LIN {X 0,Y 509.993,Z 290.092,A -85,B 0,C 180,E1 -5500.32,E2 -5500.32} C_VEL
LIN {X 0,Y 510.308,Z 281.912,A -85,B 0,C 180,E1 -5501.117,E2 -5501.117} C_VEL
LIN {X 0,Y 510.541,Z 273.397,A -85,B 0,C 180,E1 -5501.816,E2 -5501.816} C_VEL
LIN {X 0,Y 510.81,Z 263.864,A -85,B 0,C 180,E1 -5502.464,E2 -5502.464} C_VEL
LIN {X 0,Y 511.035,Z 254.914,A -85,B 0,C 180,E1 -5502.964,E2 -5502.964} C_VEL
LIN {X 0,Y 511.335,Z 244.83,A -85,B 0,C 180,E1 -5503.411,E2 -5503.411} C_VEL
LIN {X 0,Y 511.524,Z 235.312,A -85,B 0,C 180,E1 -5503.735,E2 -5503.735} C_VEL
LIN {X 0,Y 511.735,Z 224.998,A -85,B 0,C 180,E1 -5503.983,E2 -5503.983} C_VEL
LIN {X 0,Y 512.09,Z 160.549,A -85,B 0,C 180,E1 -5504.912,E2 -5504.912} C_VEL
LIN {X 0,Y 512.087,Z 131.63,A -85,B 0,C 180,E1 -5505.323,E2 -5505.323} C_VEL
LIN {X 0,Y 510.005,Z 119.074,A -85,B 0,C 180,E1 -5505.584,E2 -5505.584} C_VEL
LIN {X 0,Y 509.995,Z 117.671,A -85,B 0,C 180,E1 -5505.801,E2 -5505.801} C_VEL
LIN {X 0,Y 510.345,Z 103.483,A -85,B 0,C 180,E1 -5508.674,E2 -5508.674} C_VEL
LIN {X 0,Y 510.685,Z 89.891,A -85,B 0,C 180,E1 -5511.388,E2 -5511.388} C_VEL
LIN {X 0,Y 511.184,Z 75.466,A -85,B 0,C 180,E1 -5514.359,E2 -5514.359} C_VEL
LIN {X 0,Y 510.796,Z 71.345,A -85,B 0,C 180,E1 -5515.247,E2 -5515.247} C_VEL
LIN {X 0,Y 509.918,Z 66.493,A -85,B 0,C 180,E1 -5516.379,E2 -5516.379} C_VEL
LIN {X 0,Y 509.88,Z 66.471,A -85,B 0,C 180,E1 -5518.844,E2 -5518.844} C_VEL
LIN {X 0,Y 509.823,Z 66.48,A -85,B 0,C 180,E1 -5521.59,E2 -5521.59} C_VEL
LIN {X 0,Y 509.855,Z 66.471,A -85,B 0,C 180,E1 -5524.413,E2 -5524.413} C_VEL
LIN {X 0,Y 509.82,Z 66.479,A -85,B 0,C 180,E1 -5527.34,E2 -5527.34} C_VEL
LIN {X 0,Y 509.84,Z 66.466,A -85,B 0,C 180,E1 -5530.382,E2 -5530.382} C_VEL
LIN {X 0,Y 509.824,Z 66.478,A -85,B 0,C 180,E1 -5533.062,E2 -5533.062} C_VEL
LIN {X 0,Y 509.824,Z 66.478,A -85,B 0,C 180,E1 -5535.793,E2 -5535.793} C_VEL
LIN {X 0,Y 509.857,Z 66.471,A -85,B 0,C 180,E1 -5538.574,E2 -5538.574} C_VEL
LIN {X 0,Y 509.853,Z 66.473,A -85,B 0,C 180,E1 -5541.786,E2 -5541.786} C_VEL
LIN {X 0,Y 509.835,Z 66.474,A -85,B 0,C 180,E1 -5544.622,E2 -5544.622} C_VEL
LIN {X 0,Y 509.862,Z 66.472,A -85,B 0,C 180,E1 -5547.48,E2 -5547.48} C_VEL
LIN {X 0,Y 509.86,Z 66.471,A -85,B 0,C 180,E1 -5550.273,E2 -5550.273} C_VEL
LIN {X 0,Y 509.885,Z 66.466,A -85,B 0,C 180,E1 -5552.944,E2 -5552.944} C_VEL
LIN {X 0,Y 509.871,Z 66.468,A -85,B 0,C 180,E1 -5555.574,E2 -5555.574} C_VEL
LIN {X 0,Y 509.852,Z 66.47,A -85,B 0,C 180,E1 -5558.998,E2 -5558.998} C_VEL
LIN {X 0,Y 509.883,Z 66.459,A -85,B 0,C 180,E1 -5562.001,E2 -5562.001} C_VEL
LIN {X 0,Y 509.911,Z 66.467,A -85,B 0,C 180,E1 -5564.818,E2 -5564.818} C_VEL
LIN {X 0,Y 509.902,Z 66.468,A -85,B 0,C 180,E1 -5568.123,E2 -5568.123} C_VEL
LIN {X 0,Y 509.915,Z 66.455,A -85,B 0,C 180,E1 -5571.279,E2 -5571.279} C_VEL
LIN {X 0,Y 509.979,Z 66.455,A -85,B 0,C 180,E1 -5573.67,E2 -5573.67} C_VEL
LIN {X 0,Y 510.055,Z 66.447,A -85,B 0,C 180,E1 -5577.63,E2 -5577.63} C_VEL
LIN {X 0,Y 510.063,Z 66.436,A -85,B 0,C 180,E1 -5580.789,E2 -5580.789} C_VEL
LIN {X 0,Y 509.953,Z 66.457,A -85,B 0,C 180,E1 -5583.16,E2 -5583.16} C_VEL
LIN {X 0,Y 509.978,Z 66.455,A -85,B 0,C 180,E1 -5586.329,E2 -5586.329} C_VEL
LIN {X 0,Y 509.914,Z 66.456,A -85,B 0,C 180,E1 -5588.72,E2 -5588.72} C_VEL
LIN {X 0,Y 509.951,Z 66.46,A -85,B 0,C 180,E1 -5591.93,E2 -5591.93} C_VEL
LIN {X 0,Y 509.893,Z 66.472,A -85,B 0,C 180,E1 -5595.241,E2 -5595.241} C_VEL
LIN {X 0,Y 509.887,Z 66.46,A -85,B 0,C 180,E1 -5598,E2 -5598} C_VEL
LIN {X 0,Y 509.849,Z 66.471,A -85,B 0,C 180,E1 -5601.001,E2 -5601.001} C_VEL
LIN {X 0,Y 509.868,Z 66.47,A -85,B 0,C 180,E1 -5604.426,E2 -5604.426} C_VEL
LIN {X 0,Y 509.883,Z 66.466,A -85,B 0,C 180,E1 -5607.055,E2 -5607.055} C_VEL
LIN {X 0,Y 509.855,Z 66.471,A -85,B 0,C 180,E1 -5609.751,E2 -5609.751} C_VEL
LIN {X 0,Y 509.874,Z 66.475,A -85,B 0,C 180,E1 -5612.774,E2 -5612.774} C_VEL
LIN {X 0,Y 509.84,Z 66.471,A -85,B 0,C 180,E1 -5615.581,E2 -5615.581} C_VEL
LIN {X 0,Y 509.848,Z 66.476,A -85,B 0,C 180,E1 -5618.338,E2 -5618.338} C_VEL
LIN {X 0,Y 509.862,Z 66.468,A -85,B 0,C 180,E1 -5621.424,E2 -5621.424} C_VEL
LIN {X 0,Y 509.854,Z 66.474,A -85,B 0,C 180,E1 -5624.668,E2 -5624.668} C_VEL
LIN {X 0,Y 509.855,Z 66.46,A -85,B 0,C 180,E1 -5628.103,E2 -5628.103} C_VEL
LIN {X 0,Y 509.844,Z 66.476,A -85,B 0,C 180,E1 -5630.648,E2 -5630.648} C_VEL
LIN {X 0,Y 509.829,Z 66.474,A -85,B 0,C 180,E1 -5633.732,E2 -5633.732} C_VEL
LIN {X 0,Y 509.163,Z 66.553,A -85,B 0,C 180,E1 -5634.391,E2 -5634.391} C_VEL
LIN {X 0,Y 506.346,Z 66.901,A -85,B 0,C 180,E1 -5635.463,E2 -5635.463} C_VEL
LIN {X 0,Y 503.953,Z 67.206,A -85,B 0,C 180,E1 -5636.327,E2 -5636.327} C_VEL
LIN {X 0,Y 502.903,Z 67.336,A -85,B 0,C 180,E1 -5636.993,E2 -5636.993} C_VEL
LIN {X 0,Y 502.806,Z 67.348,A -85,B 0,C 180,E1 -5637.219,E2 -5637.219} C_VEL
LIN {X 0,Y 502.811,Z 67.347,A -85,B 0,C 180,E1 -5640.065,E2 -5640.065} C_VEL
LIN {X 0,Y 502.831,Z 67.349,A -85,B 0,C 180,E1 -5642.533,E2 -5642.533} C_VEL
LIN {X 0,Y 502.826,Z 67.35,A -85,B 0,C 180,E1 -5645.298,E2 -5645.298} C_VEL
LIN {X 0,Y 502.782,Z 67.36,A -85,B 0,C 180,E1 -5647.827,E2 -5647.827} C_VEL
LIN {X 0,Y 502.822,Z 67.35,A -85,B 0,C 180,E1 -5650.4,E2 -5650.4} C_VEL
LIN {X 0,Y 502.831,Z 67.349,A -85,B 0,C 180,E1 -5652.932,E2 -5652.932} C_VEL
LIN {X 0,Y 502.849,Z 67.352,A -85,B 0,C 180,E1 -5655.429,E2 -5655.429} C_VEL
LIN {X 0,Y 502.874,Z 67.344,A -85,B 0,C 180,E1 -5658.717,E2 -5658.717} C_VEL
LIN {X 0,Y 502.899,Z 67.341,A -85,B 0,C 180,E1 -5661.967,E2 -5661.967} C_VEL
LIN {X 0,Y 502.939,Z 67.336,A -85,B 0,C 180,E1 -5664.387,E2 -5664.387} C_VEL
LIN {X 0,Y 503.023,Z 67.327,A -85,B 0,C 180,E1 -5667.598,E2 -5667.598} C_VEL
LIN {X 0,Y 503.025,Z 67.325,A -85,B 0,C 180,E1 -5670,E2 -5670} C_VEL
LIN {X 0,Y 503.023,Z 67.326,A -85,B 0,C 180,E1 -5672.402,E2 -5672.402} C_VEL
LIN {X 0,Y 502.939,Z 67.336,A -85,B 0,C 180,E1 -5675.613,E2 -5675.613} C_VEL
LIN {X 0,Y 502.899,Z 67.341,A -85,B 0,C 180,E1 -5678.033,E2 -5678.033} C_VEL
LIN {X 0,Y 502.874,Z 67.344,A -85,B 0,C 180,E1 -5681.283,E2 -5681.283} C_VEL
LIN {X 0,Y 502.849,Z 67.352,A -85,B 0,C 180,E1 -5684.571,E2 -5684.571} C_VEL
LIN {X 0,Y 502.859,Z 67.347,A -85,B 0,C 180,E1 -5687.907,E2 -5687.907} C_VEL
LIN {X 0,Y 502.825,Z 67.354,A -85,B 0,C 180,E1 -5690.536,E2 -5690.536} C_VEL
LIN {X 0,Y 502.794,Z 67.353,A -85,B 0,C 180,E1 -5693.04,E2 -5693.04} C_VEL
LIN {X 0,Y 502.837,Z 67.349,A -85,B 0,C 180,E1 -5695.676,E2 -5695.676} C_VEL
LIN {X 0,Y 502.837,Z 67.344,A -85,B 0,C 180,E1 -5698.373,E2 -5698.373} C_VEL
LIN {X 0,Y 502.793,Z 67.353,A -85,B 0,C 180,E1 -5701.5,E2 -5701.5} C_VEL
LIN {X 0,Y 502.803,Z 67.337,A -85,B 0,C 180,E1 -5704.445,E2 -5704.445} C_VEL
LIN {X 0,Y 502.778,Z 67.353,A -85,B 0,C 180,E1 -5707.179,E2 -5707.179} C_VEL
LIN {X 0,Y 502.785,Z 67.348,A -85,B 0,C 180,E1 -5710.015,E2 -5710.015} C_VEL
LIN {X 0,Y 502.799,Z 67.336,A -85,B 0,C 180,E1 -5712.199,E2 -5712.199} C_VEL
LIN {X 0,Y 502.798,Z 67.354,A -85,B 0,C 180,E1 -5715.468,E2 -5715.468} C_VEL
LIN {X 0,Y 502.823,Z 67.348,A -85,B 0,C 180,E1 -5719.004,E2 -5719.004} C_VEL
LIN {X 0,Y 502.791,Z 67.352,A -85,B 0,C 180,E1 -5722.047,E2 -5722.047} C_VEL
LIN {X 0,Y 502.807,Z 67.35,A -85,B 0,C 180,E1 -5725.035,E2 -5725.035} C_VEL
LIN {X 0,Y 502.782,Z 67.352,A -85,B 0,C 180,E1 -5727.916,E2 -5727.916} C_VEL
LIN {X 0,Y 502.822,Z 67.351,A -85,B 0,C 180,E1 -5730.713,E2 -5730.713} C_VEL
LIN {X 0,Y 502.86,Z 67.339,A -85,B 0,C 180,E1 -5733.44,E2 -5733.44} C_VEL
LIN {X 0,Y 502.79,Z 67.351,A -85,B 0,C 180,E1 -5736.087,E2 -5736.087} C_VEL
LIN {X 0,Y 502.782,Z 67.356,A -85,B 0,C 180,E1 -5738.689,E2 -5738.689} C_VEL
LIN {X 0,Y 502.829,Z 67.339,A -85,B 0,C 180,E1 -5741.249,E2 -5741.249} C_VEL
LIN {X 0,Y 502.821,Z 67.345,A -85,B 0,C 180,E1 -5743.768,E2 -5743.768} C_VEL
LIN {X 0,Y 502.83,Z 67.351,A -85,B 0,C 180,E1 -5746.255,E2 -5746.255} C_VEL
LIN {X 0,Y 502.892,Z 67.333,A -85,B 0,C 180,E1 -5748.718,E2 -5748.718} C_VEL
LIN {X 0,Y 502.901,Z 67.333,A -85,B 0,C 180,E1 -5751.967,E2 -5751.967} C_VEL
LIN {X 0,Y 502.937,Z 67.339,A -85,B 0,C 180,E1 -5754.387,E2 -5754.387} C_VEL
LIN {X 0,Y 503.024,Z 67.321,A -85,B 0,C 180,E1 -5757.598,E2 -5757.598} C_VEL
LIN {X 0,Y 503.027,Z 67.315,A -85,B 0,C 180,E1 -5760,E2 -5760} C_VEL
LIN {X 0,Y 503.025,Z 67.322,A -85,B 0,C 180,E1 -5762.403,E2 -5762.403} C_VEL
LIN {X 0,Y 502.938,Z 67.338,A -85,B 0,C 180,E1 -5765.614,E2 -5765.614} C_VEL
LIN {X 0,Y 502.902,Z 67.333,A -85,B 0,C 180,E1 -5768.034,E2 -5768.034} C_VEL
LIN {X 0,Y 502.878,Z 67.334,A -85,B 0,C 180,E1 -5771.284,E2 -5771.284} C_VEL
LIN {X 0,Y 502.846,Z 67.343,A -85,B 0,C 180,E1 -5774.571,E2 -5774.571} C_VEL
LIN {X 0,Y 502.856,Z 67.334,A -85,B 0,C 180,E1 -5777.908,E2 -5777.908} C_VEL
LIN {X 0,Y 502.83,Z 67.341,A -85,B 0,C 180,E1 -5780.537,E2 -5780.537} C_VEL
LIN {X 0,Y 502.796,Z 67.354,A -85,B 0,C 180,E1 -5783.041,E2 -5783.041} C_VEL
LIN {X 0,Y 502.841,Z 67.34,A -85,B 0,C 180,E1 -5785.676,E2 -5785.676} C_VEL
LIN {X 0,Y 502.841,Z 67.34,A -85,B 0,C 180,E1 -5788.373,E2 -5788.373} C_VEL
LIN {X 0,Y 502.794,Z 67.352,A -85,B 0,C 180,E1 -5791.499,E2 -5791.499} C_VEL
LIN {X 0,Y 502.807,Z 67.342,A -85,B 0,C 180,E1 -5793.994,E2 -5793.994} C_VEL
LIN {X 0,Y 502.779,Z 67.356,A -85,B 0,C 180,E1 -5797.178,E2 -5797.178} C_VEL
LIN {X 0,Y 502.789,Z 67.348,A -85,B 0,C 180,E1 -5800.016,E2 -5800.016} C_VEL
LIN {X 0,Y 502.804,Z 67.352,A -85,B 0,C 180,E1 -5802.2,E2 -5802.2} C_VEL
LIN {X 0,Y 502.787,Z 67.35,A -85,B 0,C 180,E1 -5805.47,E2 -5805.47} C_VEL
LIN {X 0,Y 502.821,Z 67.341,A -85,B 0,C 180,E1 -5808.934,E2 -5808.934} C_VEL
LIN {X 0,Y 502.795,Z 67.354,A -85,B 0,C 180,E1 -5812.046,E2 -5812.046} C_VEL
LIN {X 0,Y 502.81,Z 67.347,A -85,B 0,C 180,E1 -5815.035,E2 -5815.035} C_VEL
LIN {X 0,Y 502.786,Z 67.354,A -85,B 0,C 180,E1 -5817.916,E2 -5817.916} C_VEL
LIN {X 0,Y 502.827,Z 67.35,A -85,B 0,C 180,E1 -5820.712,E2 -5820.712} C_VEL
LIN {X 0,Y 502.899,Z 67.568,A -85,B 0,C 180,E1 -5823.524,E2 -5823.524} C_VEL
LIN {X 0,Y 504.176,Z 75.331,A -85,B 0,C 180,E1 -5825.28,E2 -5825.28} C_VEL
LIN {X 0,Y 503.8,Z 87.666,A -85,B 0,C 180,E1 -5827.874,E2 -5827.874} C_VEL
LIN {X 0,Y 503.438,Z 101.167,A -85,B 0,C 180,E1 -5830.637,E2 -5830.637} C_VEL
LIN {X 0,Y 503.066,Z 114.588,A -85,B 0,C 180,E1 -5833.358,E2 -5833.358} C_VEL
LIN {X 0,Y 502.97,Z 118.697,A -85,B 0,C 180,E1 -5834.179,E2 -5834.179} C_VEL
LIN {X 0,Y 504.693,Z 129.277,A -85,B 0,C 180,E1 -5834.416,E2 -5834.416} C_VEL
LIN {X 0,Y 505.338,Z 134.211,A -85,B 0,C 180,E1 -5834.507,E2 -5834.507} C_VEL
LIN {X 0,Y 504.875,Z 223.476,A -85,B 0,C 180,E1 -5835.798,E2 -5835.798} C_VEL
LIN {X 0,Y 504.64,Z 234.247,A -85,B 0,C 180,E1 -5836.048,E2 -5836.048} C_VEL
LIN {X 0,Y 504.462,Z 243.352,A -85,B 0,C 180,E1 -5836.351,E2 -5836.351} C_VEL
LIN {X 0,Y 504.145,Z 253.716,A -85,B 0,C 180,E1 -5836.805,E2 -5836.805} C_VEL
LIN {X 0,Y 503.863,Z 263.769,A -85,B 0,C 180,E1 -5837.367,E2 -5837.367} C_VEL
LIN {X 0,Y 503.589,Z 271.853,A -85,B 0,C 180,E1 -5837.917,E2 -5837.917} C_VEL
LIN {X 0,Y 503.31,Z 280.584,A -85,B 0,C 180,E1 -5838.625,E2 -5838.625} C_VEL
LIN {X 0,Y 503.05,Z 287.981,A -85,B 0,C 180,E1 -5839.332,E2 -5839.332} C_VEL
LIN {X 0,Y 502.829,Z 295.203,A -85,B 0,C 180,E1 -5840.141,E2 -5840.141} C_VEL
LIN {X 0,Y 502.608,Z 301.404,A -85,B 0,C 180,E1 -5840.949,E2 -5840.949} C_VEL
LIN {X 0,Y 502.425,Z 307.942,A -85,B 0,C 180,E1 -5841.959,E2 -5841.959} C_VEL
LIN {X 0,Y 502.273,Z 313.495,A -85,B 0,C 180,E1 -5842.988,E2 -5842.988} C_VEL
LIN {X 0,Y 502.189,Z 317.931,A -85,B 0,C 180,E1 -5843.975,E2 -5843.975} C_VEL
LIN {X 0,Y 502.11,Z 322.251,A -85,B 0,C 180,E1 -5845.183,E2 -5845.183} C_VEL
LIN {X 0,Y 502.138,Z 324.616,A -85,B 0,C 180,E1 -5845.987,E2 -5845.987} C_VEL
LIN {X 0,Y 502.12,Z 326.411,A -85,B 0,C 180,E1 -5846.791,E2 -5846.791} C_VEL
LIN {X 0,Y 502.037,Z 328.849,A -85,B 0,C 180,E1 -5848.396,E2 -5848.396} C_VEL
LIN {X 0,Y 501.994,Z 329.435,A -85,B 0,C 180,E1 -5849.198,E2 -5849.198} C_VEL
LIN {X 0,Y 501.994,Z 329.435,A -85,B 0,C 180,E1 -5850.802,E2 -5850.802} C_VEL
LIN {X 0,Y 502.037,Z 328.849,A -85,B 0,C 180,E1 -5851.604,E2 -5851.604} C_VEL
LIN {X 0,Y 502.12,Z 326.411,A -85,B 0,C 180,E1 -5853.209,E2 -5853.209} C_VEL
LIN {X 0,Y 502.103,Z 323.466,A -85,B 0,C 180,E1 -5854.415,E2 -5854.415} C_VEL
LIN {X 0,Y 502.194,Z 319.484,A -85,B 0,C 180,E1 -5855.622,E2 -5855.622} C_VEL
LIN {X 0,Y 502.217,Z 314.548,A -85,B 0,C 180,E1 -5856.791,E2 -5856.791} C_VEL
LIN {X 0,Y 502.381,Z 309.097,A -85,B 0,C 180,E1 -5857.839,E2 -5857.839} C_VEL
LIN {X 0,Y 502.572,Z 302.781,A -85,B 0,C 180,E1 -5858.849,E2 -5858.849} C_VEL
LIN {X 0,Y 502.775,Z 296.83,A -85,B 0,C 180,E1 -5859.656,E2 -5859.656} C_VEL
LIN {X 0,Y 502.971,Z 289.9,A -85,B 0,C 180,E1 -5860.466,E2 -5860.466} C_VEL
LIN {X 0,Y 503.268,Z 281.719,A -85,B 0,C 180,E1 -5861.274,E2 -5861.274} C_VEL
LIN {X 0,Y 503.567,Z 273.206,A -85,B 0,C 180,E1 -5861.982,E2 -5861.982} C_VEL
LIN {X 0,Y 503.843,Z 264.07,A -85,B 0,C 180,E1 -5862.615,E2 -5862.615} C_VEL
LIN {X 0,Y 504.09,Z 254.723,A -85,B 0,C 180,E1 -5863.146,E2 -5863.146} C_VEL
LIN {X 0,Y 504.419,Z 244.639,A -85,B 0,C 180,E1 -5863.598,E2 -5863.598} C_VEL
LIN {X 0,Y 504.646,Z 235.122,A -85,B 0,C 180,E1 -5863.926,E2 -5863.926} C_VEL
LIN {X 0,Y 504.848,Z 224.808,A -85,B 0,C 180,E1 -5864.177,E2 -5864.177} C_VEL
LIN {X 0,Y 505.172,Z 165.727,A -85,B 0,C 180,E1 -5865.043,E2 -5865.043} C_VEL
LIN {X 0,Y 505.145,Z 131.725,A -85,B 0,C 180,E1 -5865.534,E2 -5865.534} C_VEL
LIN {X 0,Y 502.987,Z 118.974,A -85,B 0,C 180,E1 -5865.802,E2 -5865.802} C_VEL
LIN {X 0,Y 502.957,Z 117.857,A -85,B 0,C 180,E1 -5865.947,E2 -5865.947} C_VEL
LIN {X 0,Y 503.347,Z 104.398,A -85,B 0,C 180,E1 -5868.732,E2 -5868.732} C_VEL
LIN {X 0,Y 503.695,Z 90.805,A -85,B 0,C 180,E1 -5871.485,E2 -5871.485} C_VEL
LIN {X 0,Y 504.204,Z 77.414,A -85,B 0,C 180,E1 -5874.28,E2 -5874.28} C_VEL
LIN {X 0,Y 503.885,Z 72.915,A -85,B 0,C 180,E1 -5875.259,E2 -5875.259} C_VEL
LIN {X 0,Y 502.885,Z 67.367,A -85,B 0,C 180,E1 -5876.565,E2 -5876.565} C_VEL
LIN {X 0,Y 502.827,Z 67.35,A -85,B 0,C 180,E1 -5879.288,E2 -5879.288} C_VEL
LIN {X 0,Y 502.786,Z 67.355,A -85,B 0,C 180,E1 -5882.084,E2 -5882.084} C_VEL
LIN {X 0,Y 502.81,Z 67.348,A -85,B 0,C 180,E1 -5884.965,E2 -5884.965} C_VEL
LIN {X 0,Y 502.795,Z 67.354,A -85,B 0,C 180,E1 -5887.954,E2 -5887.954} C_VEL
LIN {X 0,Y 502.821,Z 67.342,A -85,B 0,C 180,E1 -5891.066,E2 -5891.066} C_VEL
LIN {X 0,Y 502.787,Z 67.351,A -85,B 0,C 180,E1 -5894.53,E2 -5894.53} C_VEL
LIN {X 0,Y 502.796,Z 67.352,A -85,B 0,C 180,E1 -5897.86,E2 -5897.86} C_VEL
LIN {X 0,Y 502.803,Z 67.351,A -85,B 0,C 180,E1 -5901.024,E2 -5901.024} C_VEL
LIN {X 0,Y 502.778,Z 67.351,A -85,B 0,C 180,E1 -5904.168,E2 -5904.168} C_VEL
LIN {X 0,Y 502.834,Z 67.347,A -85,B 0,C 180,E1 -5906.993,E2 -5906.993} C_VEL
LIN {X 0,Y 502.816,Z 67.348,A -85,B 0,C 180,E1 -5910.065,E2 -5910.065} C_VEL
LIN {X 0,Y 502.833,Z 67.344,A -85,B 0,C 180,E1 -5912.533,E2 -5912.533} C_VEL
LIN {X 0,Y 502.83,Z 67.347,A -85,B 0,C 180,E1 -5915.298,E2 -5915.298} C_VEL
LIN {X 0,Y 502.782,Z 67.351,A -85,B 0,C 180,E1 -5917.826,E2 -5917.826} C_VEL
LIN {X 0,Y 502.826,Z 67.345,A -85,B 0,C 180,E1 -5920.4,E2 -5920.4} C_VEL
LIN {X 0,Y 502.831,Z 67.345,A -85,B 0,C 180,E1 -5922.931,E2 -5922.931} C_VEL
LIN {X 0,Y 502.846,Z 67.343,A -85,B 0,C 180,E1 -5925.429,E2 -5925.429} C_VEL
LIN {X 0,Y 502.878,Z 67.334,A -85,B 0,C 180,E1 -5928.716,E2 -5928.716} C_VEL
LIN {X 0,Y 502.902,Z 67.333,A -85,B 0,C 180,E1 -5931.966,E2 -5931.966} C_VEL
LIN {X 0,Y 502.938,Z 67.338,A -85,B 0,C 180,E1 -5934.386,E2 -5934.386} C_VEL
LIN {X 0,Y 503.025,Z 67.322,A -85,B 0,C 180,E1 -5937.597,E2 -5937.597} C_VEL
LIN {X 0,Y 503.027,Z 67.315,A -85,B 0,C 180,E1 -5940,E2 -5940} C_VEL
LIN {X 0,Y 503.024,Z 67.321,A -85,B 0,C 180,E1 -5942.402,E2 -5942.402} C_VEL
LIN {X 0,Y 502.937,Z 67.339,A -85,B 0,C 180,E1 -5945.613,E2 -5945.613} C_VEL
LIN {X 0,Y 502.901,Z 67.333,A -85,B 0,C 180,E1 -5948.033,E2 -5948.033} C_VEL
LIN {X 0,Y 502.892,Z 67.333,A -85,B 0,C 180,E1 -5951.282,E2 -5951.282} C_VEL
LIN {X 0,Y 502.844,Z 67.344,A -85,B 0,C 180,E1 -5954.57,E2 -5954.57} C_VEL
LIN {X 0,Y 502.86,Z 67.335,A -85,B 0,C 180,E1 -5957.907,E2 -5957.907} C_VEL
LIN {X 0,Y 502.827,Z 67.341,A -85,B 0,C 180,E1 -5960.536,E2 -5960.536} C_VEL
LIN {X 0,Y 502.793,Z 67.356,A -85,B 0,C 180,E1 -5963.04,E2 -5963.04} C_VEL
LIN {X 0,Y 502.838,Z 67.342,A -85,B 0,C 180,E1 -5965.675,E2 -5965.675} C_VEL
LIN {X 0,Y 502.838,Z 67.34,A -85,B 0,C 180,E1 -5968.372,E2 -5968.372} C_VEL
LIN {X 0,Y 502.794,Z 67.352,A -85,B 0,C 180,E1 -5971.499,E2 -5971.499} C_VEL
LIN {X 0,Y 502.804,Z 67.348,A -85,B 0,C 180,E1 -5974.444,E2 -5974.444} C_VEL
LIN {X 0,Y 502.778,Z 67.356,A -85,B 0,C 180,E1 -5977.178,E2 -5977.178} C_VEL
LIN {X 0,Y 502.814,Z 67.347,A -85,B 0,C 180,E1 -5980.012,E2 -5980.012} C_VEL
LIN {X 0,Y 502.77,Z 67.355,A -85,B 0,C 180,E1 -5983.231,E2 -5983.231} C_VEL
LIN {X 0,Y 502.786,Z 67.348,A -85,B 0,C 180,E1 -5985.661,E2 -5985.661} C_VEL
LIN {X 0,Y 502.816,Z 67.341,A -85,B 0,C 180,E1 -5989.005,E2 -5989.005} C_VEL
LIN {X 0,Y 502.791,Z 67.357,A -85,B 0,C 180,E1 -5992.046,E2 -5992.046} C_VEL
LIN {X 0,Y 502.807,Z 67.338,A -85,B 0,C 180,E1 -5995.035,E2 -5995.035} C_VEL
LIN {X 0,Y 502.806,Z 67.348,A -85,B 0,C 180,E1 -5997.219,E2 -5997.219} C_VEL
LIN {X 0,Y 502.104,Z 67.443,A -85,B 0,C 180,E1 -5997.888,E2 -5997.888} C_VEL
LIN {X 0,Y 499.239,Z 67.794,A -85,B 0,C 180,E1 -5998.973,E2 -5998.973} C_VEL
LIN {X 0,Y 496.844,Z 68.093,A -85,B 0,C 180,E1 -5999.848,E2 -5999.848} C_VEL
LIN {X 0,Y 495.828,Z 68.213,A -85,B 0,C 180,E1 -6000.524,E2 -6000.524} C_VEL
LIN {X 0,Y 495.75,Z 68.221,A -85,B 0,C 180,E1 -6000.753,E2 -6000.753} C_VEL
LIN {X 0,Y 495.82,Z 68.222,A -85,B 0,C 180,E1 -6003.251,E2 -6003.251} C_VEL
LIN {X 0,Y 495.75,Z 68.236,A -85,B 0,C 180,E1 -6005.725,E2 -6005.725} C_VEL
LIN {X 0,Y 495.741,Z 68.232,A -85,B 0,C 180,E1 -6008.371,E2 -6008.371} C_VEL
LIN {X 0,Y 495.781,Z 68.227,A -85,B 0,C 180,E1 -6010.972,E2 -6010.972} C_VEL
LIN {X 0,Y 495.776,Z 68.233,A -85,B 0,C 180,E1 -6013.53,E2 -6013.53} C_VEL
LIN {X 0,Y 495.795,Z 68.226,A -85,B 0,C 180,E1 -6016.056,E2 -6016.056} C_VEL
LIN {X 0,Y 495.849,Z 68.219,A -85,B 0,C 180,E1 -6018.555,E2 -6018.555} C_VEL
LIN {X 0,Y 495.87,Z 68.218,A -85,B 0,C 180,E1 -6021.852,E2 -6021.852} C_VEL
LIN {X 0,Y 495.896,Z 68.213,A -85,B 0,C 180,E1 -6024.307,E2 -6024.307} C_VEL
LIN {X 0,Y 495.991,Z 68.203,A -85,B 0,C 180,E1 -6027.564,E2 -6027.564} C_VEL
LIN {X 0,Y 495.996,Z 68.201,A -85,B 0,C 180,E1 -6030,E2 -6030} C_VEL
LIN {X 0,Y 495.991,Z 68.203,A -85,B 0,C 180,E1 -6032.436,E2 -6032.436} C_VEL
LIN {X 0,Y 495.896,Z 68.213,A -85,B 0,C 180,E1 -6035.693,E2 -6035.693} C_VEL
LIN {X 0,Y 495.87,Z 68.218,A -85,B 0,C 180,E1 -6038.148,E2 -6038.148} C_VEL
LIN {X 0,Y 495.849,Z 68.219,A -85,B 0,C 180,E1 -6041.445,E2 -6041.445} C_VEL
LIN {X 0,Y 495.791,Z 68.23,A -85,B 0,C 180,E1 -6044.783,E2 -6044.783} C_VEL
LIN {X 0,Y 495.783,Z 68.226,A -85,B 0,C 180,E1 -6047.319,E2 -6047.319} C_VEL
LIN {X 0,Y 495.775,Z 68.23,A -85,B 0,C 180,E1 -6049.89,E2 -6049.89} C_VEL
LIN {X 0,Y 495.762,Z 68.23,A -85,B 0,C 180,E1 -6052.863,E2 -6052.863} C_VEL
LIN {X 0,Y 495.788,Z 68.231,A -85,B 0,C 180,E1 -6056.068,E2 -6056.068} C_VEL
LIN {X 0,Y 495.769,Z 68.22,A -85,B 0,C 180,E1 -6058.815,E2 -6058.815} C_VEL
LIN {X 0,Y 495.756,Z 68.233,A -85,B 0,C 180,E1 -6061.726,E2 -6061.726} C_VEL
LIN {X 0,Y 495.773,Z 68.211,A -85,B 0,C 180,E1 -6064.695,E2 -6064.695} C_VEL
LIN {X 0,Y 495.729,Z 68.236,A -85,B 0,C 180,E1 -6067.562,E2 -6067.562} C_VEL
LIN {X 0,Y 495.763,Z 68.218,A -85,B 0,C 180,E1 -6070.7,E2 -6070.7} C_VEL
LIN {X 0,Y 495.729,Z 68.229,A -85,B 0,C 180,E1 -6074.001,E2 -6074.001} C_VEL
LIN {X 0,Y 495.723,Z 68.236,A -85,B 0,C 180,E1 -6077.117,E2 -6077.117} C_VEL
LIN {X 0,Y 495.782,Z 68.223,A -85,B 0,C 180,E1 -6079.95,E2 -6079.95} C_VEL
LIN {X 0,Y 495.728,Z 68.232,A -85,B 0,C 180,E1 -6082.553,E2 -6082.553} C_VEL
LIN {X 0,Y 495.783,Z 68.223,A -85,B 0,C 180,E1 -6085.458,E2 -6085.458} C_VEL
LIN {X 0,Y 495.754,Z 68.228,A -85,B 0,C 180,E1 -6088.364,E2 -6088.364} C_VEL
LIN {X 0,Y 495.786,Z 68.219,A -85,B 0,C 180,E1 -6091.507,E2 -6091.507} C_VEL
LIN {X 0,Y 495.789,Z 68.218,A -85,B 0,C 180,E1 -6093.933,E2 -6093.933} C_VEL
LIN {X 0,Y 495.76,Z 68.23,A -85,B 0,C 180,E1 -6097.139,E2 -6097.139} C_VEL
LIN {X 0,Y 495.77,Z 68.221,A -85,B 0,C 180,E1 -6100.11,E2 -6100.11} C_VEL
LIN {X 0,Y 495.786,Z 68.224,A -85,B 0,C 180,E1 -6102.682,E2 -6102.682} C_VEL
LIN {X 0,Y 495.789,Z 68.224,A -85,B 0,C 180,E1 -6105.218,E2 -6105.218} C_VEL
LIN {X 0,Y 495.867,Z 68.21,A -85,B 0,C 180,E1 -6108.556,E2 -6108.556} C_VEL
LIN {X 0,Y 495.872,Z 68.207,A -85,B 0,C 180,E1 -6111.852,E2 -6111.852} C_VEL
LIN {X 0,Y 495.895,Z 68.217,A -85,B 0,C 180,E1 -6114.307,E2 -6114.307} C_VEL
LIN {X 0,Y 495.993,Z 68.197,A -85,B 0,C 180,E1 -6117.564,E2 -6117.564} C_VEL
LIN {X 0,Y 495.983,Z 68.19,A -85,B 0,C 180,E1 -6120.812,E2 -6120.812} C_VEL
LIN {X 0,Y 495.993,Z 68.198,A -85,B 0,C 180,E1 -6122.437,E2 -6122.437} C_VEL
LIN {X 0,Y 495.896,Z 68.216,A -85,B 0,C 180,E1 -6125.694,E2 -6125.694} C_VEL
LIN {X 0,Y 495.873,Z 68.206,A -85,B 0,C 180,E1 -6128.148,E2 -6128.148} C_VEL
LIN {X 0,Y 495.852,Z 68.211,A -85,B 0,C 180,E1 -6131.446,E2 -6131.446} C_VEL
LIN {X 0,Y 495.791,Z 68.222,A -85,B 0,C 180,E1 -6134.783,E2 -6134.783} C_VEL
LIN {X 0,Y 495.783,Z 68.224,A -85,B 0,C 180,E1 -6137.319,E2 -6137.319} C_VEL
LIN {X 0,Y 495.772,Z 68.222,A -85,B 0,C 180,E1 -6139.891,E2 -6139.891} C_VEL
LIN {X 0,Y 495.763,Z 68.228,A -85,B 0,C 180,E1 -6142.862,E2 -6142.862} C_VEL
LIN {X 0,Y 495.792,Z 68.216,A -85,B 0,C 180,E1 -6146.068,E2 -6146.068} C_VEL
LIN {X 0,Y 495.773,Z 68.224,A -85,B 0,C 180,E1 -6148.815,E2 -6148.815} C_VEL
LIN {X 0,Y 495.756,Z 68.227,A -85,B 0,C 180,E1 -6151.726,E2 -6151.726} C_VEL
LIN {X 0,Y 495.773,Z 68.223,A -85,B 0,C 180,E1 -6154.695,E2 -6154.695} C_VEL
LIN {X 0,Y 495.731,Z 68.231,A -85,B 0,C 180,E1 -6157.562,E2 -6157.562} C_VEL
LIN {X 0,Y 495.768,Z 68.228,A -85,B 0,C 180,E1 -6160.7,E2 -6160.7} C_VEL
LIN {X 0,Y 495.729,Z 68.232,A -85,B 0,C 180,E1 -6164.002,E2 -6164.002} C_VEL
LIN {X 0,Y 495.727,Z 68.232,A -85,B 0,C 180,E1 -6167.117,E2 -6167.117} C_VEL
LIN {X 0,Y 495.76,Z 68.221,A -85,B 0,C 180,E1 -6169.953,E2 -6169.953} C_VEL
LIN {X 0,Y 495.732,Z 68.235,A -85,B 0,C 180,E1 -6172.553,E2 -6172.553} C_VEL
LIN {X 0,Y 495.786,Z 68.222,A -85,B 0,C 180,E1 -6175.458,E2 -6175.458} C_VEL
LIN {X 0,Y 495.758,Z 68.231,A -85,B 0,C 180,E1 -6178.364,E2 -6178.364} C_VEL
LIN {X 0,Y 495.791,Z 68.229,A -85,B 0,C 180,E1 -6181.507,E2 -6181.507} C_VEL
LIN {X 0,Y 495.813,Z 68.256,A -85,B 0,C 180,E1 -6183.254,E2 -6183.254} C_VEL
LIN {X 0,Y 497.203,Z 76.259,A -85,B 0,C 180,E1 -6185.133,E2 -6185.133} C_VEL
LIN {X 0,Y 496.953,Z 85.726,A -85,B 0,C 180,E1 -6187.173,E2 -6187.173} C_VEL
LIN {X 0,Y 496.433,Z 102.038,A -85,B 0,C 180,E1 -6190.568,E2 -6190.568} C_VEL
LIN {X 0,Y 495.988,Z 116.376,A -85,B 0,C 180,E1 -6193.537,E2 -6193.537} C_VEL
LIN {X 0,Y 495.941,Z 118.399,A -85,B 0,C 180,E1 -6193.938,E2 -6193.938} C_VEL
LIN {X 0,Y 496.765,Z 123.524,A -85,B 0,C 180,E1 -6194.08,E2 -6194.08} C_VEL
LIN {X 0,Y 498.484,Z 134.02,A -85,B 0,C 180,E1 -6194.289,E2 -6194.289} C_VEL
LIN {X 0,Y 497.992,Z 223.286,A -85,B 0,C 180,E1 -6195.597,E2 -6195.597} C_VEL
LIN {X 0,Y 497.786,Z 233.183,A -85,B 0,C 180,E1 -6195.826,E2 -6195.826} C_VEL
LIN {X 0,Y 497.57,Z 243.161,A -85,B 0,C 180,E1 -6196.159,E2 -6196.159} C_VEL
LIN {X 0,Y 497.21,Z 253.525,A -85,B 0,C 180,E1 -6196.617,E2 -6196.617} C_VEL
LIN {X 0,Y 496.944,Z 262.767,A -85,B 0,C 180,E1 -6197.136,E2 -6197.136} C_VEL
LIN {X 0,Y 496.623,Z 271.662,A -85,B 0,C 180,E1 -6197.744,E2 -6197.744} C_VEL
LIN {X 0,Y 496.344,Z 280.394,A -85,B 0,C 180,E1 -6198.463,E2 -6198.463} C_VEL
LIN {X 0,Y 496.052,Z 287.79,A -85,B 0,C 180,E1 -6199.18,E2 -6199.18} C_VEL
LIN {X 0,Y 495.802,Z 295.011,A -85,B 0,C 180,E1 -6200,E2 -6200} C_VEL
LIN {X 0,Y 495.555,Z 301.213,A -85,B 0,C 180,E1 -6200.819,E2 -6200.819} C_VEL
LIN {X 0,Y 495.375,Z 307.751,A -85,B 0,C 180,E1 -6201.844,E2 -6201.844} C_VEL
LIN {X 0,Y 495.261,Z 312.252,A -85,B 0,C 180,E1 -6202.662,E2 -6202.662} C_VEL
LIN {X 0,Y 495.101,Z 317.346,A -85,B 0,C 180,E1 -6203.785,E2 -6203.785} C_VEL
LIN {X 0,Y 495.102,Z 320.823,A -85,B 0,C 180,E1 -6204.706,E2 -6204.706} C_VEL
LIN {X 0,Y 495.032,Z 324.425,A -85,B 0,C 180,E1 -6205.929,E2 -6205.929} C_VEL
LIN {X 0,Y 495.042,Z 326.221,A -85,B 0,C 180,E1 -6206.745,E2 -6206.745} C_VEL
LIN {X 0,Y 494.963,Z 328.659,A -85,B 0,C 180,E1 -6208.373,E2 -6208.373} C_VEL
LIN {X 0,Y 494.914,Z 329.245,A -85,B 0,C 180,E1 -6209.186,E2 -6209.186} C_VEL
LIN {X 0,Y 494.914,Z 329.245,A -85,B 0,C 180,E1 -6210.814,E2 -6210.814} C_VEL
LIN {X 0,Y 494.963,Z 328.659,A -85,B 0,C 180,E1 -6211.627,E2 -6211.627} C_VEL
LIN {X 0,Y 495.042,Z 326.221,A -85,B 0,C 180,E1 -6213.255,E2 -6213.255} C_VEL
LIN {X 0,Y 495.009,Z 323.275,A -85,B 0,C 180,E1 -6214.479,E2 -6214.479} C_VEL
LIN {X 0,Y 495.109,Z 319.293,A -85,B 0,C 180,E1 -6215.703,E2 -6215.703} C_VEL
LIN {X 0,Y 495.131,Z 316.08,A -85,B 0,C 180,E1 -6216.52,E2 -6216.52} C_VEL
LIN {X 0,Y 495.295,Z 310.061,A -85,B 0,C 180,E1 -6217.747,E2 -6217.747} C_VEL
LIN {X 0,Y 495.498,Z 303.966,A -85,B 0,C 180,E1 -6218.77,E2 -6218.77} C_VEL
LIN {X 0,Y 495.688,Z 298.265,A -85,B 0,C 180,E1 -6219.59,E2 -6219.59} C_VEL
LIN {X 0,Y 495.961,Z 289.709,A -85,B 0,C 180,E1 -6220.615,E2 -6220.615} C_VEL
LIN {X 0,Y 496.28,Z 281.528,A -85,B 0,C 180,E1 -6221.435,E2 -6221.435} C_VEL
LIN {X 0,Y 496.601,Z 273.015,A -85,B 0,C 180,E1 -6222.152,E2 -6222.152} C_VEL
LIN {X 0,Y 496.887,Z 264.335,A -85,B 0,C 180,E1 -6222.765,E2 -6222.765} C_VEL
LIN {X 0,Y 497.169,Z 254.532,A -85,B 0,C 180,E1 -6223.332,E2 -6223.332} C_VEL
LIN {X 0,Y 497.518,Z 244.449,A -85,B 0,C 180,E1 -6223.791,E2 -6223.791} C_VEL
LIN {X 0,Y 497.77,Z 234.932,A -85,B 0,C 180,E1 -6224.122,E2 -6224.122} C_VEL
LIN {X 0,Y 497.969,Z 224.617,A -85,B 0,C 180,E1 -6224.377,E2 -6224.377} C_VEL
LIN {X 0,Y 498.377,Z 158.042,A -85,B 0,C 180,E1 -6225.363,E2 -6225.363} C_VEL
LIN {X 0,Y 498.359,Z 132.886,A -85,B 0,C 180,E1 -6225.732,E2 -6225.732} C_VEL
LIN {X 0,Y 495.955,Z 118.635,A -85,B 0,C 180,E1 -6226.042,E2 -6226.042} C_VEL
LIN {X 0,Y 495.936,Z 117.82,A -85,B 0,C 180,E1 -6226.148,E2 -6226.148} C_VEL
LIN {X 0,Y 496.327,Z 105.982,A -85,B 0,C 180,E1 -6228.654,E2 -6228.654} C_VEL
LIN {X 0,Y 496.714,Z 91.72,A -85,B 0,C 180,E1 -6231.584,E2 -6231.584} C_VEL
LIN {X 0,Y 497.258,Z 78.302,A -85,B 0,C 180,E1 -6234.419,E2 -6234.419} C_VEL
LIN {X 0,Y 496.712,Z 73.188,A -85,B 0,C 180,E1 -6235.565,E2 -6235.565} C_VEL
LIN {X 0,Y 495.84,Z 68.243,A -85,B 0,C 180,E1 -6236.752,E2 -6236.752} C_VEL
LIN {X 0,Y 495.769,Z 68.229,A -85,B 0,C 180,E1 -6239.746,E2 -6239.746} C_VEL
LIN {X 0,Y 495.77,Z 68.227,A -85,B 0,C 180,E1 -6242.594,E2 -6242.594} C_VEL
LIN {X 0,Y 495.758,Z 68.227,A -85,B 0,C 180,E1 -6245.537,E2 -6245.537} C_VEL
LIN {X 0,Y 495.765,Z 68.225,A -85,B 0,C 180,E1 -6248.768,E2 -6248.768} C_VEL
LIN {X 0,Y 495.758,Z 68.232,A -85,B 0,C 180,E1 -6251.781,E2 -6251.781} C_VEL
LIN {X 0,Y 495.739,Z 68.233,A -85,B 0,C 180,E1 -6255.14,E2 -6255.14} C_VEL
LIN {X 0,Y 495.757,Z 68.227,A -85,B 0,C 180,E1 -6258.218,E2 -6258.218} C_VEL
LIN {X 0,Y 495.752,Z 68.234,A -85,B 0,C 180,E1 -6261.408,E2 -6261.408} C_VEL
LIN {X 0,Y 495.751,Z 68.227,A -85,B 0,C 180,E1 -6264.462,E2 -6264.462} C_VEL
LIN {X 0,Y 495.768,Z 68.228,A -85,B 0,C 180,E1 -6267.405,E2 -6267.405} C_VEL
LIN {X 0,Y 495.767,Z 68.227,A -85,B 0,C 180,E1 -6270.253,E2 -6270.253} C_VEL
LIN {X 0,Y 495.824,Z 68.215,A -85,B 0,C 180,E1 -6273.25,E2 -6273.25} C_VEL
LIN {X 0,Y 495.753,Z 68.226,A -85,B 0,C 180,E1 -6275.725,E2 -6275.725} C_VEL
LIN {X 0,Y 495.744,Z 68.232,A -85,B 0,C 180,E1 -6278.371,E2 -6278.371} C_VEL
LIN {X 0,Y 495.785,Z 68.215,A -85,B 0,C 180,E1 -6280.971,E2 -6280.971} C_VEL
LIN {X 0,Y 495.779,Z 68.22,A -85,B 0,C 180,E1 -6283.53,E2 -6283.53} C_VEL
LIN {X 0,Y 495.794,Z 68.225,A -85,B 0,C 180,E1 -6286.055,E2 -6286.055} C_VEL
LIN {X 0,Y 495.852,Z 68.211,A -85,B 0,C 180,E1 -6288.554,E2 -6288.554} C_VEL
LIN {X 0,Y 495.873,Z 68.206,A -85,B 0,C 180,E1 -6291.852,E2 -6291.852} C_VEL
LIN {X 0,Y 495.896,Z 68.216,A -85,B 0,C 180,E1 -6294.306,E2 -6294.306} C_VEL
LIN {X 0,Y 495.993,Z 68.198,A -85,B 0,C 180,E1 -6297.563,E2 -6297.563} C_VEL
LIN {X 0,Y 495.983,Z 68.189,A -85,B 0,C 180,E1 -6300.811,E2 -6300.811} C_VEL
LIN {X 0,Y 495.993,Z 68.197,A -85,B 0,C 180,E1 -6302.436,E2 -6302.436} C_VEL
LIN {X 0,Y 495.895,Z 68.217,A -85,B 0,C 180,E1 -6305.693,E2 -6305.693} C_VEL
LIN {X 0,Y 495.872,Z 68.207,A -85,B 0,C 180,E1 -6308.148,E2 -6308.148} C_VEL
LIN {X 0,Y 495.867,Z 68.21,A -85,B 0,C 180,E1 -6311.444,E2 -6311.444} C_VEL
LIN {X 0,Y 495.789,Z 68.224,A -85,B 0,C 180,E1 -6314.782,E2 -6314.782} C_VEL
LIN {X 0,Y 495.786,Z 68.224,A -85,B 0,C 180,E1 -6317.318,E2 -6317.318} C_VEL
LIN {X 0,Y 495.77,Z 68.221,A -85,B 0,C 180,E1 -6319.89,E2 -6319.89} C_VEL
LIN {X 0,Y 495.76,Z 68.23,A -85,B 0,C 180,E1 -6322.861,E2 -6322.861} C_VEL
LIN {X 0,Y 495.789,Z 68.218,A -85,B 0,C 180,E1 -6326.067,E2 -6326.067} C_VEL
LIN {X 0,Y 495.77,Z 68.225,A -85,B 0,C 180,E1 -6328.814,E2 -6328.814} C_VEL
LIN {X 0,Y 495.756,Z 68.228,A -85,B 0,C 180,E1 -6331.726,E2 -6331.726} C_VEL
LIN {X 0,Y 495.774,Z 68.224,A -85,B 0,C 180,E1 -6334.695,E2 -6334.695} C_VEL
LIN {X 0,Y 495.729,Z 68.232,A -85,B 0,C 180,E1 -6337.561,E2 -6337.561} C_VEL
LIN {X 0,Y 495.775,Z 68.226,A -85,B 0,C 180,E1 -6340.698,E2 -6340.698} C_VEL
LIN {X 0,Y 495.731,Z 68.233,A -85,B 0,C 180,E1 -6344.001,E2 -6344.001} C_VEL
LIN {X 0,Y 495.722,Z 68.216,A -85,B 0,C 180,E1 -6347.117,E2 -6347.117} C_VEL
LIN {X 0,Y 495.756,Z 68.223,A -85,B 0,C 180,E1 -6349.953,E2 -6349.953} C_VEL
LIN {X 0,Y 495.728,Z 68.234,A -85,B 0,C 180,E1 -6352.552,E2 -6352.552} C_VEL
LIN {X 0,Y 495.782,Z 68.214,A -85,B 0,C 180,E1 -6355.457,E2 -6355.457} C_VEL
LIN {X 0,Y 495.753,Z 68.232,A -85,B 0,C 180,E1 -6358.364,E2 -6358.364} C_VEL
LIN {X 0,Y 495.75,Z 68.221,A -85,B 0,C 180,E1 -6360.753,E2 -6360.753} C_VEL
LIN {X 0,Y 495.092,Z 68.307,A -85,B 0,C 180,E1 -6361.432,E2 -6361.432} C_VEL
LIN {X 0,Y 492.236,Z 68.669,A -85,B 0,C 180,E1 -6362.534,E2 -6362.534} C_VEL
LIN {X 0,Y 489.828,Z 68.97,A -85,B 0,C 180,E1 -6363.423,E2 -6363.423} C_VEL
LIN {X 0,Y 488.812,Z 69.099,A -85,B 0,C 180,E1 -6364.109,E2 -6364.109} C_VEL
LIN {X 0,Y 488.739,Z 69.104,A -85,B 0,C 180,E1 -6364.342,E2 -6364.342} C_VEL
LIN {X 0,Y 488.725,Z 69.107,A -85,B 0,C 180,E1 -6367.153,E2 -6367.153} C_VEL
LIN {X 0,Y 488.725,Z 69.111,A -85,B 0,C 180,E1 -6369.811,E2 -6369.811} C_VEL
LIN {X 0,Y 488.731,Z 69.105,A -85,B 0,C 180,E1 -6372.423,E2 -6372.423} C_VEL
LIN {X 0,Y 488.762,Z 69.104,A -85,B 0,C 180,E1 -6375,E2 -6375} C_VEL
LIN {X 0,Y 488.802,Z 69.097,A -85,B 0,C 180,E1 -6378.388,E2 -6378.388} C_VEL
LIN {X 0,Y 488.815,Z 69.098,A -85,B 0,C 180,E1 -6381.734,E2 -6381.734} C_VEL
LIN {X 0,Y 488.856,Z 69.09,A -85,B 0,C 180,E1 -6384.224,E2 -6384.224} C_VEL
LIN {X 0,Y 488.959,Z 69.08,A -85,B 0,C 180,E1 -6387.529,E2 -6387.529} C_VEL
LIN {X 0,Y 488.951,Z 69.082,A -85,B 0,C 180,E1 -6390.824,E2 -6390.824} C_VEL
LIN {X 0,Y 488.959,Z 69.079,A -85,B 0,C 180,E1 -6392.471,E2 -6392.471} C_VEL
LIN {X 0,Y 488.856,Z 69.09,A -85,B 0,C 180,E1 -6395.776,E2 -6395.776} C_VEL
LIN {X 0,Y 488.815,Z 69.098,A -85,B 0,C 180,E1 -6398.266,E2 -6398.266} C_VEL
LIN {X 0,Y 488.802,Z 69.096,A -85,B 0,C 180,E1 -6401.612,E2 -6401.612} C_VEL
LIN {X 0,Y 488.762,Z 69.104,A -85,B 0,C 180,E1 -6405,E2 -6405} C_VEL
LIN {X 0,Y 488.752,Z 69.108,A -85,B 0,C 180,E1 -6408.442,E2 -6408.442} C_VEL
LIN {X 0,Y 488.704,Z 69.109,A -85,B 0,C 180,E1 -6411.071,E2 -6411.071} C_VEL
LIN {X 0,Y 488.691,Z 69.112,A -85,B 0,C 180,E1 -6413.745,E2 -6413.745} C_VEL
LIN {X 0,Y 488.789,Z 69.097,A -85,B 0,C 180,E1 -6416.944,E2 -6416.944} C_VEL
LIN {X 0,Y 488.707,Z 69.109,A -85,B 0,C 180,E1 -6420.363,E2 -6420.363} C_VEL
LIN {X 0,Y 488.732,Z 69.104,A -85,B 0,C 180,E1 -6423.485,E2 -6423.485} C_VEL
LIN {X 0,Y 488.686,Z 69.109,A -85,B 0,C 180,E1 -6426.356,E2 -6426.356} C_VEL
LIN {X 0,Y 488.698,Z 69.11,A -85,B 0,C 180,E1 -6429.254,E2 -6429.254} C_VEL
LIN {X 0,Y 488.703,Z 69.093,A -85,B 0,C 180,E1 -6431.6,E2 -6431.6} C_VEL
LIN {X 0,Y 488.708,Z 69.102,A -85,B 0,C 180,E1 -6434.802,E2 -6434.802} C_VEL
LIN {X 0,Y 488.688,Z 69.113,A -85,B 0,C 180,E1 -6437.475,E2 -6437.475} C_VEL
LIN {X 0,Y 488.73,Z 69.104,A -85,B 0,C 180,E1 -6439.677,E2 -6439.677} C_VEL
LIN {X 0,Y 488.676,Z 69.11,A -85,B 0,C 180,E1 -6442.278,E2 -6442.278} C_VEL
LIN {X 0,Y 488.726,Z 69.103,A -85,B 0,C 180,E1 -6445.052,E2 -6445.052} C_VEL
LIN {X 0,Y 488.701,Z 69.106,A -85,B 0,C 180,E1 -6448.046,E2 -6448.046} C_VEL
LIN {X 0,Y 488.721,Z 69.108,A -85,B 0,C 180,E1 -6450.73,E2 -6450.73} C_VEL
LIN {X 0,Y 488.755,Z 69.095,A -85,B 0,C 180,E1 -6453.529,E2 -6453.529} C_VEL
LIN {X 0,Y 488.691,Z 69.109,A -85,B 0,C 180,E1 -6456.255,E2 -6456.255} C_VEL
LIN {X 0,Y 488.744,Z 69.097,A -85,B 0,C 180,E1 -6459.176,E2 -6459.176} C_VEL
LIN {X 0,Y 488.733,Z 69.098,A -85,B 0,C 180,E1 -6462.424,E2 -6462.424} C_VEL
LIN {X 0,Y 488.761,Z 69.101,A -85,B 0,C 180,E1 -6465,E2 -6465} C_VEL
LIN {X 0,Y 488.829,Z 69.089,A -85,B 0,C 180,E1 -6468.389,E2 -6468.389} C_VEL
LIN {X 0,Y 488.816,Z 69.084,A -85,B 0,C 180,E1 -6471.734,E2 -6471.734} C_VEL
LIN {X 0,Y 488.854,Z 69.094,A -85,B 0,C 180,E1 -6474.225,E2 -6474.225} C_VEL
LIN {X 0,Y 488.961,Z 69.072,A -85,B 0,C 180,E1 -6477.529,E2 -6477.529} C_VEL
LIN {X 0,Y 488.934,Z 69.068,A -85,B 0,C 180,E1 -6480.824,E2 -6480.824} C_VEL
LIN {X 0,Y 488.961,Z 69.074,A -85,B 0,C 180,E1 -6482.472,E2 -6482.472} C_VEL
LIN {X 0,Y 488.855,Z 69.094,A -85,B 0,C 180,E1 -6485.776,E2 -6485.776} C_VEL
LIN {X 0,Y 488.817,Z 69.084,A -85,B 0,C 180,E1 -6488.267,E2 -6488.267} C_VEL
LIN {X 0,Y 488.806,Z 69.091,A -85,B 0,C 180,E1 -6491.613,E2 -6491.613} C_VEL
LIN {X 0,Y 488.763,Z 69.099,A -85,B 0,C 180,E1 -6495.001,E2 -6495.001} C_VEL
LIN {X 0,Y 488.756,Z 69.087,A -85,B 0,C 180,E1 -6498.443,E2 -6498.443} C_VEL
LIN {X 0,Y 488.708,Z 69.104,A -85,B 0,C 180,E1 -6501.071,E2 -6501.071} C_VEL
LIN {X 0,Y 488.694,Z 69.108,A -85,B 0,C 180,E1 -6503.746,E2 -6503.746} C_VEL
LIN {X 0,Y 488.793,Z 69.091,A -85,B 0,C 180,E1 -6506.944,E2 -6506.944} C_VEL
LIN {X 0,Y 488.711,Z 69.106,A -85,B 0,C 180,E1 -6510.363,E2 -6510.363} C_VEL
LIN {X 0,Y 488.736,Z 69.096,A -85,B 0,C 180,E1 -6513.485,E2 -6513.485} C_VEL
LIN {X 0,Y 488.684,Z 69.109,A -85,B 0,C 180,E1 -6516.355,E2 -6516.355} C_VEL
LIN {X 0,Y 488.703,Z 69.104,A -85,B 0,C 180,E1 -6519.255,E2 -6519.255} C_VEL
LIN {X 0,Y 488.708,Z 69.105,A -85,B 0,C 180,E1 -6521.6,E2 -6521.6} C_VEL
LIN {X 0,Y 488.703,Z 69.109,A -85,B 0,C 180,E1 -6524.803,E2 -6524.803} C_VEL
LIN {X 0,Y 488.693,Z 69.107,A -85,B 0,C 180,E1 -6527.475,E2 -6527.475} C_VEL
LIN {X 0,Y 488.735,Z 69.094,A -85,B 0,C 180,E1 -6529.677,E2 -6529.677} C_VEL
LIN {X 0,Y 488.684,Z 69.11,A -85,B 0,C 180,E1 -6532.842,E2 -6532.842} C_VEL
LIN {X 0,Y 488.736,Z 69.104,A -85,B 0,C 180,E1 -6535.888,E2 -6535.888} C_VEL
LIN {X 0,Y 488.695,Z 69.111,A -85,B 0,C 180,E1 -6538.821,E2 -6538.821} C_VEL
LIN {X 0,Y 488.748,Z 69.108,A -85,B 0,C 180,E1 -6541.672,E2 -6541.672} C_VEL
LIN {X 0,Y 488.809,Z 69.331,A -85,B 0,C 180,E1 -6543.147,E2 -6543.147} C_VEL
LIN {X 0,Y 490.249,Z 77.432,A -85,B 0,C 180,E1 -6545.046,E2 -6545.046} C_VEL
LIN {X 0,Y 489.943,Z 87.389,A -85,B 0,C 180,E1 -6547.213,E2 -6547.213} C_VEL
LIN {X 0,Y 489.426,Z 102.909,A -85,B 0,C 180,E1 -6550.497,E2 -6550.497} C_VEL
LIN {X 0,Y 488.987,Z 116.195,A -85,B 0,C 180,E1 -6553.295,E2 -6553.295} C_VEL
LIN {X 0,Y 488.956,Z 118.324,A -85,B 0,C 180,E1 -6553.712,E2 -6553.712} C_VEL
LIN {X 0,Y 490.384,Z 127.177,A -85,B 0,C 180,E1 -6553.924,E2 -6553.924} C_VEL
LIN {X 0,Y 491.644,Z 135.801,A -85,B 0,C 180,E1 -6554.094,E2 -6554.094} C_VEL
LIN {X 0,Y 491.114,Z 223.095,A -85,B 0,C 180,E1 -6555.391,E2 -6555.391} C_VEL
LIN {X 0,Y 490.909,Z 232.992,A -85,B 0,C 180,E1 -6555.623,E2 -6555.623} C_VEL
LIN {X 0,Y 490.687,Z 242.971,A -85,B 0,C 180,E1 -6555.96,E2 -6555.96} C_VEL
LIN {X 0,Y 490.302,Z 253.334,A -85,B 0,C 180,E1 -6556.425,E2 -6556.425} C_VEL
LIN {X 0,Y 490.019,Z 262.475,A -85,B 0,C 180,E1 -6556.945,E2 -6556.945} C_VEL
LIN {X 0,Y 489.646,Z 271.47,A -85,B 0,C 180,E1 -6557.567,E2 -6557.567} C_VEL
LIN {X 0,Y 489.376,Z 280.203,A -85,B 0,C 180,E1 -6558.296,E2 -6558.296} C_VEL
LIN {X 0,Y 489.067,Z 287.599,A -85,B 0,C 180,E1 -6559.024,E2 -6559.024} C_VEL
LIN {X 0,Y 488.776,Z 294.82,A -85,B 0,C 180,E1 -6559.855,E2 -6559.855} C_VEL
LIN {X 0,Y 488.516,Z 301.021,A -85,B 0,C 180,E1 -6560.686,E2 -6560.686} C_VEL
LIN {X 0,Y 488.313,Z 307.559,A -85,B 0,C 180,E1 -6561.725,E2 -6561.725} C_VEL
LIN {X 0,Y 488.185,Z 312.06,A -85,B 0,C 180,E1 -6562.556,E2 -6562.556} C_VEL
LIN {X 0,Y 488.003,Z 317.61,A -85,B 0,C 180,E1 -6563.816,E2 -6563.816} C_VEL
LIN {X 0,Y 487.966,Z 321.87,A -85,B 0,C 180,E1 -6565.043,E2 -6565.043} C_VEL
LIN {X 0,Y 487.928,Z 324.233,A -85,B 0,C 180,E1 -6565.87,E2 -6565.87} C_VEL
LIN {X 0,Y 487.965,Z 326.031,A -85,B 0,C 180,E1 -6566.697,E2 -6566.697} C_VEL
LIN {X 0,Y 487.891,Z 328.469,A -85,B 0,C 180,E1 -6568.349,E2 -6568.349} C_VEL
LIN {X 0,Y 487.837,Z 329.055,A -85,B 0,C 180,E1 -6569.175,E2 -6569.175} C_VEL
LIN {X 0,Y 487.837,Z 329.055,A -85,B 0,C 180,E1 -6570.825,E2 -6570.825} C_VEL
LIN {X 0,Y 487.891,Z 328.469,A -85,B 0,C 180,E1 -6571.651,E2 -6571.651} C_VEL
LIN {X 0,Y 487.965,Z 326.031,A -85,B 0,C 180,E1 -6573.303,E2 -6573.303} C_VEL
LIN {X 0,Y 487.921,Z 323.085,A -85,B 0,C 180,E1 -6574.544,E2 -6574.544} C_VEL
LIN {X 0,Y 488.008,Z 319.102,A -85,B 0,C 180,E1 -6575.786,E2 -6575.786} C_VEL
LIN {X 0,Y 488.044,Z 315.889,A -85,B 0,C 180,E1 -6576.615,E2 -6576.615} C_VEL
LIN {X 0,Y 488.22,Z 309.869,A -85,B 0,C 180,E1 -6577.86,E2 -6577.86} C_VEL
LIN {X 0,Y 488.431,Z 303.774,A -85,B 0,C 180,E1 -6578.898,E2 -6578.898} C_VEL
LIN {X 0,Y 488.658,Z 298.074,A -85,B 0,C 180,E1 -6579.729,E2 -6579.729} C_VEL
LIN {X 0,Y 488.964,Z 289.518,A -85,B 0,C 180,E1 -6580.769,E2 -6580.769} C_VEL
LIN {X 0,Y 489.305,Z 281.337,A -85,B 0,C 180,E1 -6581.6,E2 -6581.6} C_VEL
LIN {X 0,Y 489.628,Z 272.823,A -85,B 0,C 180,E1 -6582.328,E2 -6582.328} C_VEL
LIN {X 0,Y 489.942,Z 264.109,A -85,B 0,C 180,E1 -6582.952,E2 -6582.952} C_VEL
LIN {X 0,Y 490.253,Z 254.341,A -85,B 0,C 180,E1 -6583.524,E2 -6583.524} C_VEL
LIN {X 0,Y 490.614,Z 244.258,A -85,B 0,C 180,E1 -6583.989,E2 -6583.989} C_VEL
LIN {X 0,Y 490.866,Z 234.741,A -85,B 0,C 180,E1 -6584.325,E2 -6584.325} C_VEL
LIN {X 0,Y 491.108,Z 224.427,A -85,B 0,C 180,E1 -6584.583,E2 -6584.583} C_VEL
LIN {X 0,Y 491.549,Z 155.817,A -85,B 0,C 180,E1 -6585.612,E2 -6585.612} C_VEL
LIN {X 0,Y 491.447,Z 133.188,A -85,B 0,C 180,E1 -6585.951,E2 -6585.951} C_VEL
LIN {X 0,Y 488.94,Z 118.453,A -85,B 0,C 180,E1 -6586.278,E2 -6586.278} C_VEL
LIN {X 0,Y 488.928,Z 117.633,A -85,B 0,C 180,E1 -6586.386,E2 -6586.386} C_VEL
LIN {X 0,Y 489.305,Z 106.144,A -85,B 0,C 180,E1 -6588.863,E2 -6588.863} C_VEL
LIN {X 0,Y 489.712,Z 93.684,A -85,B 0,C 180,E1 -6591.466,E2 -6591.466} C_VEL
LIN {X 0,Y 490.311,Z 79.189,A -85,B 0,C 180,E1 -6594.562,E2 -6594.562} C_VEL
LIN {X 0,Y 489.49,Z 73.046,A -85,B 0,C 180,E1 -6595.971,E2 -6595.971} C_VEL
LIN {X 0,Y 488.803,Z 69.12,A -85,B 0,C 180,E1 -6596.945,E2 -6596.945} C_VEL
LIN {X 0,Y 488.712,Z 69.111,A -85,B 0,C 180,E1 -6600.363,E2 -6600.363} C_VEL
LIN {X 0,Y 488.738,Z 69.107,A -85,B 0,C 180,E1 -6603.484,E2 -6603.484} C_VEL
LIN {X 0,Y 488.69,Z 69.109,A -85,B 0,C 180,E1 -6606.355,E2 -6606.355} C_VEL
LIN {X 0,Y 488.703,Z 69.106,A -85,B 0,C 180,E1 -6609.254,E2 -6609.254} C_VEL
LIN {X 0,Y 488.708,Z 69.106,A -85,B 0,C 180,E1 -6611.599,E2 -6611.599} C_VEL
LIN {X 0,Y 488.703,Z 69.106,A -85,B 0,C 180,E1 -6614.802,E2 -6614.802} C_VEL
LIN {X 0,Y 488.693,Z 69.114,A -85,B 0,C 180,E1 -6617.474,E2 -6617.474} C_VEL
LIN {X 0,Y 488.734,Z 69.101,A -85,B 0,C 180,E1 -6619.676,E2 -6619.676} C_VEL
LIN {X 0,Y 488.681,Z 69.113,A -85,B 0,C 180,E1 -6622.841,E2 -6622.841} C_VEL
LIN {X 0,Y 488.733,Z 69.095,A -85,B 0,C 180,E1 -6625.887,E2 -6625.887} C_VEL
LIN {X 0,Y 488.693,Z 69.112,A -85,B 0,C 180,E1 -6628.82,E2 -6628.82} C_VEL
LIN {X 0,Y 488.745,Z 69.095,A -85,B 0,C 180,E1 -6631.671,E2 -6631.671} C_VEL
LIN {X 0,Y 488.749,Z 69.096,A -85,B 0,C 180,E1 -6634.444,E2 -6634.444} C_VEL
LIN {X 0,Y 488.725,Z 69.105,A -85,B 0,C 180,E1 -6637.153,E2 -6637.153} C_VEL
LIN {X 0,Y 488.726,Z 69.097,A -85,B 0,C 180,E1 -6639.81,E2 -6639.81} C_VEL
LIN {X 0,Y 488.73,Z 69.097,A -85,B 0,C 180,E1 -6642.423,E2 -6642.423} C_VEL
LIN {X 0,Y 488.763,Z 69.099,A -85,B 0,C 180,E1 -6644.999,E2 -6644.999} C_VEL
LIN {X 0,Y 488.806,Z 69.091,A -85,B 0,C 180,E1 -6648.387,E2 -6648.387} C_VEL
LIN {X 0,Y 488.817,Z 69.084,A -85,B 0,C 180,E1 -6651.733,E2 -6651.733} C_VEL
LIN {X 0,Y 488.855,Z 69.094,A -85,B 0,C 180,E1 -6654.224,E2 -6654.224} C_VEL
LIN {X 0,Y 488.961,Z 69.074,A -85,B 0,C 180,E1 -6657.528,E2 -6657.528} C_VEL
LIN {X 0,Y 488.934,Z 69.066,A -85,B 0,C 180,E1 -6660.823,E2 -6660.823} C_VEL
LIN {X 0,Y 488.961,Z 69.072,A -85,B 0,C 180,E1 -6662.471,E2 -6662.471} C_VEL
LIN {X 0,Y 488.854,Z 69.094,A -85,B 0,C 180,E1 -6665.775,E2 -6665.775} C_VEL
LIN {X 0,Y 488.816,Z 69.084,A -85,B 0,C 180,E1 -6668.266,E2 -6668.266} C_VEL
LIN {X 0,Y 488.829,Z 69.089,A -85,B 0,C 180,E1 -6671.611,E2 -6671.611} C_VEL
LIN {X 0,Y 488.761,Z 69.101,A -85,B 0,C 180,E1 -6675,E2 -6675} C_VEL
LIN {X 0,Y 488.754,Z 69.09,A -85,B 0,C 180,E1 -6678.442,E2 -6678.442} C_VEL
LIN {X 0,Y 488.705,Z 69.105,A -85,B 0,C 180,E1 -6681.07,E2 -6681.07} C_VEL
LIN {X 0,Y 488.691,Z 69.109,A -85,B 0,C 180,E1 -6683.745,E2 -6683.745} C_VEL
LIN {X 0,Y 488.79,Z 69.092,A -85,B 0,C 180,E1 -6686.943,E2 -6686.943} C_VEL
LIN {X 0,Y 488.708,Z 69.106,A -85,B 0,C 180,E1 -6690.363,E2 -6690.363} C_VEL
LIN {X 0,Y 488.733,Z 69.098,A -85,B 0,C 180,E1 -6693.484,E2 -6693.484} C_VEL
LIN {X 0,Y 488.686,Z 69.108,A -85,B 0,C 180,E1 -6696.355,E2 -6696.355} C_VEL
LIN {X 0,Y 488.735,Z 69.101,A -85,B 0,C 180,E1 -6699.25,E2 -6699.25} C_VEL
LIN {X 0,Y 488.709,Z 69.103,A -85,B 0,C 180,E1 -6701.6,E2 -6701.6} C_VEL
LIN {X 0,Y 488.709,Z 69.105,A -85,B 0,C 180,E1 -6704.801,E2 -6704.801} C_VEL
LIN {X 0,Y 488.688,Z 69.091,A -85,B 0,C 180,E1 -6707.474,E2 -6707.474} C_VEL
LIN {X 0,Y 488.729,Z 69.095,A -85,B 0,C 180,E1 -6709.676,E2 -6709.676} C_VEL
LIN {X 0,Y 488.679,Z 69.109,A -85,B 0,C 180,E1 -6712.841,E2 -6712.841} C_VEL
LIN {X 0,Y 488.732,Z 69.094,A -85,B 0,C 180,E1 -6715.887,E2 -6715.887} C_VEL
LIN {X 0,Y 488.689,Z 69.108,A -85,B 0,C 180,E1 -6718.82,E2 -6718.82} C_VEL
LIN {X 0,Y 488.742,Z 69.099,A -85,B 0,C 180,E1 -6721.671,E2 -6721.671} C_VEL
LIN {X 0,Y 488.739,Z 69.104,A -85,B 0,C 180,E1 -6724.342,E2 -6724.342} C_VEL
LIN {X 0,Y 488.095,Z 69.187,A -85,B 0,C 180,E1 -6725.029,E2 -6725.029} C_VEL
LIN {X 0,Y 485.229,Z 69.549,A -85,B 0,C 180,E1 -6726.146,E2 -6726.146} C_VEL
LIN {X 0,Y 482.784,Z 69.853,A -85,B 0,C 180,E1 -6727.045,E2 -6727.045} C_VEL
LIN {X 0,Y 481.725,Z 69.983,A -85,B 0,C 180,E1 -6727.741,E2 -6727.741} C_VEL
LIN {X 0,Y 481.635,Z 69.991,A -85,B 0,C 180,E1 -6727.976,E2 -6727.976} C_VEL
LIN {X 0,Y 481.704,Z 69.981,A -85,B 0,C 180,E1 -6730.393,E2 -6730.393} C_VEL
LIN {X 0,Y 481.688,Z 69.984,A -85,B 0,C 180,E1 -6733.034,E2 -6733.034} C_VEL
LIN {X 0,Y 481.691,Z 69.987,A -85,B 0,C 180,E1 -6735.639,E2 -6735.639} C_VEL
LIN {X 0,Y 481.748,Z 69.976,A -85,B 0,C 180,E1 -6738.215,E2 -6738.215} C_VEL
LIN {X 0,Y 481.76,Z 69.977,A -85,B 0,C 180,E1 -6741.612,E2 -6741.612} C_VEL
LIN {X 0,Y 481.816,Z 69.967,A -85,B 0,C 180,E1 -6744.14,E2 -6744.14} C_VEL
LIN {X 0,Y 481.926,Z 69.956,A -85,B 0,C 180,E1 -6747.493,E2 -6747.493} C_VEL
LIN {X 0,Y 481.902,Z 69.96,A -85,B 0,C 180,E1 -6750.836,E2 -6750.836} C_VEL
LIN {X 0,Y 481.926,Z 69.956,A -85,B 0,C 180,E1 -6752.507,E2 -6752.507} C_VEL
LIN {X 0,Y 481.816,Z 69.967,A -85,B 0,C 180,E1 -6755.86,E2 -6755.86} C_VEL
LIN {X 0,Y 481.76,Z 69.977,A -85,B 0,C 180,E1 -6758.388,E2 -6758.388} C_VEL
LIN {X 0,Y 481.748,Z 69.976,A -85,B 0,C 180,E1 -6761.785,E2 -6761.785} C_VEL
LIN {X 0,Y 481.741,Z 69.977,A -85,B 0,C 180,E1 -6765.224,E2 -6765.224} C_VEL
LIN {X 0,Y 481.709,Z 69.983,A -85,B 0,C 180,E1 -6768.722,E2 -6768.722} C_VEL
LIN {X 0,Y 481.643,Z 69.988,A -85,B 0,C 180,E1 -6771.395,E2 -6771.395} C_VEL
LIN {X 0,Y 481.674,Z 69.989,A -85,B 0,C 180,E1 -6774.113,E2 -6774.113} C_VEL
LIN {X 0,Y 481.744,Z 69.975,A -85,B 0,C 180,E1 -6777.139,E2 -6777.139} C_VEL
LIN {X 0,Y 481.675,Z 69.977,A -85,B 0,C 180,E1 -6779.741,E2 -6779.741} C_VEL
LIN {X 0,Y 481.67,Z 69.982,A -85,B 0,C 180,E1 -6782.674,E2 -6782.674} C_VEL
LIN {X 0,Y 481.64,Z 69.978,A -85,B 0,C 180,E1 -6785.709,E2 -6785.709} C_VEL
LIN {X 0,Y 481.668,Z 69.983,A -85,B 0,C 180,E1 -6788.859,E2 -6788.859} C_VEL
LIN {X 0,Y 481.648,Z 69.968,A -85,B 0,C 180,E1 -6791.913,E2 -6791.913} C_VEL
LIN {X 0,Y 481.656,Z 69.979,A -85,B 0,C 180,E1 -6794.458,E2 -6794.458} C_VEL
LIN {X 0,Y 481.646,Z 69.985,A -85,B 0,C 180,E1 -6797.84,E2 -6797.84} C_VEL
LIN {X 0,Y 481.707,Z 69.975,A -85,B 0,C 180,E1 -6800.647,E2 -6800.647} C_VEL
LIN {X 0,Y 481.64,Z 69.983,A -85,B 0,C 180,E1 -6804.291,E2 -6804.291} C_VEL
LIN {X 0,Y 481.67,Z 69.987,A -85,B 0,C 180,E1 -6807.326,E2 -6807.326} C_VEL
LIN {X 0,Y 481.676,Z 69.981,A -85,B 0,C 180,E1 -6810.259,E2 -6810.259} C_VEL
LIN {X 0,Y 481.744,Z 69.97,A -85,B 0,C 180,E1 -6813.113,E2 -6813.113} C_VEL
LIN {X 0,Y 481.675,Z 69.981,A -85,B 0,C 180,E1 -6815.887,E2 -6815.887} C_VEL
LIN {X 0,Y 481.701,Z 69.975,A -85,B 0,C 180,E1 -6819.028,E2 -6819.028} C_VEL
LIN {X 0,Y 481.706,Z 69.969,A -85,B 0,C 180,E1 -6822.159,E2 -6822.159} C_VEL
LIN {X 0,Y 481.741,Z 69.978,A -85,B 0,C 180,E1 -6824.776,E2 -6824.776} C_VEL
LIN {X 0,Y 481.794,Z 69.968,A -85,B 0,C 180,E1 -6828.217,E2 -6828.217} C_VEL
LIN {X 0,Y 481.762,Z 69.962,A -85,B 0,C 180,E1 -6831.612,E2 -6831.612} C_VEL
LIN {X 0,Y 481.815,Z 69.969,A -85,B 0,C 180,E1 -6834.14,E2 -6834.14} C_VEL
LIN {X 0,Y 481.927,Z 69.948,A -85,B 0,C 180,E1 -6837.493,E2 -6837.493} C_VEL
LIN {X 0,Y 481.886,Z 69.945,A -85,B 0,C 180,E1 -6840.836,E2 -6840.836} C_VEL
LIN {X 0,Y 481.928,Z 69.949,A -85,B 0,C 180,E1 -6842.508,E2 -6842.508} C_VEL
LIN {X 0,Y 481.816,Z 69.969,A -85,B 0,C 180,E1 -6845.861,E2 -6845.861} C_VEL
LIN {X 0,Y 481.763,Z 69.961,A -85,B 0,C 180,E1 -6848.389,E2 -6848.389} C_VEL
LIN {X 0,Y 481.751,Z 69.972,A -85,B 0,C 180,E1 -6851.785,E2 -6851.785} C_VEL
LIN {X 0,Y 481.743,Z 69.976,A -85,B 0,C 180,E1 -6855.225,E2 -6855.225} C_VEL
LIN {X 0,Y 481.713,Z 69.964,A -85,B 0,C 180,E1 -6858.722,E2 -6858.722} C_VEL
LIN {X 0,Y 481.647,Z 69.988,A -85,B 0,C 180,E1 -6861.395,E2 -6861.395} C_VEL
LIN {X 0,Y 481.678,Z 69.98,A -85,B 0,C 180,E1 -6864.113,E2 -6864.113} C_VEL
LIN {X 0,Y 481.748,Z 69.968,A -85,B 0,C 180,E1 -6867.14,E2 -6867.14} C_VEL
LIN {X 0,Y 481.68,Z 69.981,A -85,B 0,C 180,E1 -6869.741,E2 -6869.741} C_VEL
LIN {X 0,Y 481.673,Z 69.985,A -85,B 0,C 180,E1 -6872.675,E2 -6872.675} C_VEL
LIN {X 0,Y 481.639,Z 69.984,A -85,B 0,C 180,E1 -6875.71,E2 -6875.71} C_VEL
LIN {X 0,Y 481.673,Z 69.984,A -85,B 0,C 180,E1 -6878.859,E2 -6878.859} C_VEL
LIN {X 0,Y 481.654,Z 69.984,A -85,B 0,C 180,E1 -6881.913,E2 -6881.913} C_VEL
LIN {X 0,Y 481.656,Z 69.987,A -85,B 0,C 180,E1 -6884.458,E2 -6884.458} C_VEL
LIN {X 0,Y 481.649,Z 69.986,A -85,B 0,C 180,E1 -6887.84,E2 -6887.84} C_VEL
LIN {X 0,Y 481.663,Z 69.981,A -85,B 0,C 180,E1 -6890.654,E2 -6890.654} C_VEL
LIN {X 0,Y 481.632,Z 69.987,A -85,B 0,C 180,E1 -6893.376,E2 -6893.376} C_VEL
LIN {X 0,Y 481.712,Z 69.984,A -85,B 0,C 180,E1 -6896.33,E2 -6896.33} C_VEL
LIN {X 0,Y 481.653,Z 69.989,A -85,B 0,C 180,E1 -6899.418,E2 -6899.418} C_VEL
LIN {X 0,Y 481.712,Z 69.98,A -85,B 0,C 180,E1 -6902.559,E2 -6902.559} C_VEL
LIN {X 0,Y 481.788,Z 70.214,A -85,B 0,C 180,E1 -6902.952,E2 -6902.952} C_VEL
LIN {X 0,Y 483.301,Z 79.055,A -85,B 0,C 180,E1 -6905.058,E2 -6905.058} C_VEL
LIN {X 0,Y 482.875,Z 90.331,A -85,B 0,C 180,E1 -6907.539,E2 -6907.539} C_VEL
LIN {X 0,Y 482.348,Z 104.812,A -85,B 0,C 180,E1 -6910.642,E2 -6910.642} C_VEL
LIN {X 0,Y 481.947,Z 117.3,A -85,B 0,C 180,E1 -6913.338,E2 -6913.338} C_VEL
LIN {X 0,Y 481.957,Z 118.298,A -85,B 0,C 180,E1 -6913.481,E2 -6913.481} C_VEL
LIN {X 0,Y 484.727,Z 135.169,A -85,B 0,C 180,E1 -6913.854,E2 -6913.854} C_VEL
LIN {X 0,Y 484.251,Z 222.905,A -85,B 0,C 180,E1 -6915.179,E2 -6915.179} C_VEL
LIN {X 0,Y 484.043,Z 232.802,A -85,B 0,C 180,E1 -6915.415,E2 -6915.415} C_VEL
LIN {X 0,Y 483.793,Z 242.78,A -85,B 0,C 180,E1 -6915.756,E2 -6915.756} C_VEL
LIN {X 0,Y 483.408,Z 253.144,A -85,B 0,C 180,E1 -6916.228,E2 -6916.228} C_VEL
LIN {X 0,Y 483.095,Z 262.284,A -85,B 0,C 180,E1 -6916.754,E2 -6916.754} C_VEL
LIN {X 0,Y 482.688,Z 271.279,A -85,B 0,C 180,E1 -6917.385,E2 -6917.385} C_VEL
LIN {X 0,Y 482.406,Z 280.04,A -85,B 0,C 180,E1 -6918.127,E2 -6918.127} C_VEL
LIN {X 0,Y 482.069,Z 287.408,A -85,B 0,C 180,E1 -6918.862,E2 -6918.862} C_VEL
LIN {X 0,Y 481.738,Z 294.628,A -85,B 0,C 180,E1 -6919.705,E2 -6919.705} C_VEL
LIN {X 0,Y 481.472,Z 300.83,A -85,B 0,C 180,E1 -6920.548,E2 -6920.548} C_VEL
LIN {X 0,Y 481.263,Z 307.368,A -85,B 0,C 180,E1 -6921.603,E2 -6921.603} C_VEL
LIN {X 0,Y 481.1,Z 311.869,A -85,B 0,C 180,E1 -6922.445,E2 -6922.445} C_VEL
LIN {X 0,Y 480.937,Z 316.828,A -85,B 0,C 180,E1 -6923.564,E2 -6923.564} C_VEL
LIN {X 0,Y 480.923,Z 320.441,A -85,B 0,C 180,E1 -6924.549,E2 -6924.549} C_VEL
LIN {X 0,Y 480.828,Z 324.042,A -85,B 0,C 180,E1 -6925.809,E2 -6925.809} C_VEL
LIN {X 0,Y 480.888,Z 325.84,A -85,B 0,C 180,E1 -6926.649,E2 -6926.649} C_VEL
LIN {X 0,Y 480.793,Z 328.278,A -85,B 0,C 180,E1 -6928.325,E2 -6928.325} C_VEL
LIN {X 0,Y 480.763,Z 328.865,A -85,B 0,C 180,E1 -6929.162,E2 -6929.162} C_VEL
LIN {X 0,Y 480.763,Z 328.865,A -85,B 0,C 180,E1 -6930.838,E2 -6930.838} C_VEL
LIN {X 0,Y 480.793,Z 328.278,A -85,B 0,C 180,E1 -6931.675,E2 -6931.675} C_VEL
LIN {X 0,Y 480.888,Z 325.84,A -85,B 0,C 180,E1 -6933.351,E2 -6933.351} C_VEL
LIN {X 0,Y 480.839,Z 322.894,A -85,B 0,C 180,E1 -6934.611,E2 -6934.611} C_VEL
LIN {X 0,Y 480.911,Z 318.91,A -85,B 0,C 180,E1 -6935.871,E2 -6935.871} C_VEL
LIN {X 0,Y 481.02,Z 313.783,A -85,B 0,C 180,E1 -6937.134,E2 -6937.134} C_VEL
LIN {X 0,Y 481.22,Z 308.523,A -85,B 0,C 180,E1 -6938.186,E2 -6938.186} C_VEL
LIN {X 0,Y 481.415,Z 302.206,A -85,B 0,C 180,E1 -6939.241,E2 -6939.241} C_VEL
LIN {X 0,Y 481.658,Z 296.255,A -85,B 0,C 180,E1 -6940.084,E2 -6940.084} C_VEL
LIN {X 0,Y 481.981,Z 289.327,A -85,B 0,C 180,E1 -6940.927,E2 -6940.927} C_VEL
LIN {X 0,Y 482.333,Z 281.146,A -85,B 0,C 180,E1 -6941.77,E2 -6941.77} C_VEL
LIN {X 0,Y 482.604,Z 274.014,A -85,B 0,C 180,E1 -6942.401,E2 -6942.401} C_VEL
LIN {X 0,Y 483.025,Z 263.918,A -85,B 0,C 180,E1 -6943.14,E2 -6943.14} C_VEL
LIN {X 0,Y 483.362,Z 254.151,A -85,B 0,C 180,E1 -6943.72,E2 -6943.72} C_VEL
LIN {X 0,Y 483.744,Z 244.068,A -85,B 0,C 180,E1 -6944.192,E2 -6944.192} C_VEL
LIN {X 0,Y 484.007,Z 234.551,A -85,B 0,C 180,E1 -6944.533,E2 -6944.533} C_VEL
LIN {X 0,Y 484.24,Z 224.237,A -85,B 0,C 180,E1 -6944.794,E2 -6944.794} C_VEL
LIN {X 0,Y 484.69,Z 161.493,A -85,B 0,C 180,E1 -6945.75,E2 -6945.75} C_VEL
LIN {X 0,Y 484.647,Z 134.203,A -85,B 0,C 180,E1 -6946.163,E2 -6946.163} C_VEL
LIN {X 0,Y 481.93,Z 118.339,A -85,B 0,C 180,E1 -6946.517,E2 -6946.517} C_VEL
LIN {X 0,Y 481.916,Z 117.445,A -85,B 0,C 180,E1 -6946.631,E2 -6946.631} C_VEL
LIN {X 0,Y 482.39,Z 105.005,A -85,B 0,C 180,E1 -6949.357,E2 -6949.357} C_VEL
LIN {X 0,Y 482.897,Z 90.411,A -85,B 0,C 180,E1 -6952.46,E2 -6952.46} C_VEL
LIN {X 0,Y 483.334,Z 80.076,A -85,B 0,C 180,E1 -6954.711,E2 -6954.711} C_VEL
LIN {X 0,Y 482.282,Z 72.909,A -85,B 0,C 180,E1 -6956.389,E2 -6956.389} C_VEL
LIN {X 0,Y 481.756,Z 69.999,A -85,B 0,C 180,E1 -6957.14,E2 -6957.14} C_VEL
LIN {X 0,Y 481.682,Z 69.983,A -85,B 0,C 180,E1 -6959.741,E2 -6959.741} C_VEL
LIN {X 0,Y 481.675,Z 69.983,A -85,B 0,C 180,E1 -6962.674,E2 -6962.674} C_VEL
LIN {X 0,Y 481.644,Z 69.985,A -85,B 0,C 180,E1 -6965.709,E2 -6965.709} C_VEL
LIN {X 0,Y 481.673,Z 69.981,A -85,B 0,C 180,E1 -6968.859,E2 -6968.859} C_VEL
LIN {X 0,Y 481.654,Z 69.988,A -85,B 0,C 180,E1 -6971.912,E2 -6971.912} C_VEL
LIN {X 0,Y 481.656,Z 69.983,A -85,B 0,C 180,E1 -6974.458,E2 -6974.458} C_VEL
LIN {X 0,Y 481.649,Z 69.987,A -85,B 0,C 180,E1 -6977.839,E2 -6977.839} C_VEL
LIN {X 0,Y 481.663,Z 69.98,A -85,B 0,C 180,E1 -6980.654,E2 -6980.654} C_VEL
LIN {X 0,Y 481.629,Z 69.99,A -85,B 0,C 180,E1 -6983.376,E2 -6983.376} C_VEL
LIN {X 0,Y 481.711,Z 69.969,A -85,B 0,C 180,E1 -6986.33,E2 -6986.33} C_VEL
LIN {X 0,Y 481.652,Z 69.987,A -85,B 0,C 180,E1 -6989.417,E2 -6989.417} C_VEL
LIN {X 0,Y 481.701,Z 69.973,A -85,B 0,C 180,E1 -6992.168,E2 -6992.168} C_VEL
LIN {X 0,Y 481.719,Z 69.98,A -85,B 0,C 180,E1 -6994.97,E2 -6994.97} C_VEL
LIN {X 0,Y 481.651,Z 69.983,A -85,B 0,C 180,E1 -6997.704,E2 -6997.704} C_VEL
LIN {X 0,Y 481.706,Z 69.973,A -85,B 0,C 180,E1 -7000.393,E2 -7000.393} C_VEL
LIN {X 0,Y 481.689,Z 69.977,A -85,B 0,C 180,E1 -7003.033,E2 -7003.033} C_VEL
LIN {X 0,Y 481.69,Z 69.979,A -85,B 0,C 180,E1 -7005.638,E2 -7005.638} C_VEL
LIN {X 0,Y 481.751,Z 69.972,A -85,B 0,C 180,E1 -7008.215,E2 -7008.215} C_VEL
LIN {X 0,Y 481.763,Z 69.961,A -85,B 0,C 180,E1 -7011.611,E2 -7011.611} C_VEL
LIN {X 0,Y 481.816,Z 69.969,A -85,B 0,C 180,E1 -7014.139,E2 -7014.139} C_VEL
LIN {X 0,Y 481.928,Z 69.949,A -85,B 0,C 180,E1 -7017.492,E2 -7017.492} C_VEL
LIN {X 0,Y 481.886,Z 69.944,A -85,B 0,C 180,E1 -7020.835,E2 -7020.835} C_VEL
LIN {X 0,Y 481.927,Z 69.948,A -85,B 0,C 180,E1 -7022.507,E2 -7022.507} C_VEL
LIN {X 0,Y 481.815,Z 69.969,A -85,B 0,C 180,E1 -7025.86,E2 -7025.86} C_VEL
LIN {X 0,Y 481.762,Z 69.962,A -85,B 0,C 180,E1 -7028.388,E2 -7028.388} C_VEL
LIN {X 0,Y 481.794,Z 69.968,A -85,B 0,C 180,E1 -7031.783,E2 -7031.783} C_VEL
LIN {X 0,Y 481.741,Z 69.978,A -85,B 0,C 180,E1 -7035.224,E2 -7035.224} C_VEL
LIN {X 0,Y 481.711,Z 69.968,A -85,B 0,C 180,E1 -7038.721,E2 -7038.721} C_VEL
LIN {X 0,Y 481.645,Z 69.989,A -85,B 0,C 180,E1 -7041.394,E2 -7041.394} C_VEL
LIN {X 0,Y 481.675,Z 69.981,A -85,B 0,C 180,E1 -7044.113,E2 -7044.113} C_VEL
LIN {X 0,Y 481.745,Z 69.968,A -85,B 0,C 180,E1 -7047.139,E2 -7047.139} C_VEL
LIN {X 0,Y 481.677,Z 69.981,A -85,B 0,C 180,E1 -7049.741,E2 -7049.741} C_VEL
LIN {X 0,Y 481.671,Z 69.987,A -85,B 0,C 180,E1 -7052.674,E2 -7052.674} C_VEL
LIN {X 0,Y 481.64,Z 69.983,A -85,B 0,C 180,E1 -7055.709,E2 -7055.709} C_VEL
LIN {X 0,Y 481.707,Z 69.975,A -85,B 0,C 180,E1 -7059.353,E2 -7059.353} C_VEL
LIN {X 0,Y 481.646,Z 69.985,A -85,B 0,C 180,E1 -7062.16,E2 -7062.16} C_VEL
LIN {X 0,Y 481.656,Z 69.979,A -85,B 0,C 180,E1 -7065.542,E2 -7065.542} C_VEL
LIN {X 0,Y 481.653,Z 69.977,A -85,B 0,C 180,E1 -7068.958,E2 -7068.958} C_VEL
LIN {X 0,Y 481.653,Z 69.989,A -85,B 0,C 180,E1 -7071.992,E2 -7071.992} C_VEL
LIN {X 0,Y 481.69,Z 69.967,A -85,B 0,C 180,E1 -7075.318,E2 -7075.318} C_VEL
LIN {X 0,Y 481.642,Z 69.99,A -85,B 0,C 180,E1 -7078.312,E2 -7078.312} C_VEL
LIN {X 0,Y 481.697,Z 69.973,A -85,B 0,C 180,E1 -7081.218,E2 -7081.218} C_VEL
LIN {X 0,Y 481.698,Z 69.986,A -85,B 0,C 180,E1 -7084.043,E2 -7084.043} C_VEL
LIN {X 0,Y 481.671,Z 69.984,A -85,B 0,C 180,E1 -7086.812,E2 -7086.812} C_VEL
LIN {X 0,Y 481.635,Z 69.991,A -85,B 0,C 180,E1 -7087.976,E2 -7087.976} C_VEL
LIN {X 0,Y 480.966,Z 70.073,A -85,B 0,C 180,E1 -7088.674,E2 -7088.674} C_VEL
LIN {X 0,Y 478.138,Z 70.429,A -85,B 0,C 180,E1 -7089.809,E2 -7089.809} C_VEL
LIN {X 0,Y 475.754,Z 70.726,A -85,B 0,C 180,E1 -7090.723,E2 -7090.723} C_VEL
LIN {X 0,Y 474.734,Z 70.853,A -85,B 0,C 180,E1 -7091.429,E2 -7091.429} C_VEL
LIN {X 0,Y 474.652,Z 70.863,A -85,B 0,C 180,E1 -7091.668,E2 -7091.668} C_VEL
LIN {X 0,Y 474.697,Z 70.854,A -85,B 0,C 180,E1 -7094.544,E2 -7094.544} C_VEL
LIN {X 0,Y 474.701,Z 70.855,A -85,B 0,C 180,E1 -7098.038,E2 -7098.038} C_VEL
LIN {X 0,Y 474.725,Z 70.854,A -85,B 0,C 180,E1 -7101.486,E2 -7101.486} C_VEL
LIN {X 0,Y 474.778,Z 70.844,A -85,B 0,C 180,E1 -7104.052,E2 -7104.052} C_VEL
LIN {X 0,Y 474.891,Z 70.833,A -85,B 0,C 180,E1 -7107.455,E2 -7107.455} C_VEL
LIN {X 0,Y 474.909,Z 70.828,A -85,B 0,C 180,E1 -7110,E2 -7110} C_VEL
LIN {X 0,Y 474.891,Z 70.833,A -85,B 0,C 180,E1 -7112.545,E2 -7112.545} C_VEL
LIN {X 0,Y 474.778,Z 70.844,A -85,B 0,C 180,E1 -7115.948,E2 -7115.948} C_VEL
LIN {X 0,Y 474.725,Z 70.854,A -85,B 0,C 180,E1 -7118.514,E2 -7118.514} C_VEL
LIN {X 0,Y 474.701,Z 70.855,A -85,B 0,C 180,E1 -7121.962,E2 -7121.962} C_VEL
LIN {X 0,Y 474.697,Z 70.854,A -85,B 0,C 180,E1 -7125.456,E2 -7125.456} C_VEL
LIN {X 0,Y 474.662,Z 70.859,A -85,B 0,C 180,E1 -7129.01,E2 -7129.01} C_VEL
LIN {X 0,Y 474.587,Z 70.869,A -85,B 0,C 180,E1 -7131.729,E2 -7131.729} C_VEL
LIN {X 0,Y 474.656,Z 70.862,A -85,B 0,C 180,E1 -7134.493,E2 -7134.493} C_VEL
LIN {X 0,Y 474.696,Z 70.853,A -85,B 0,C 180,E1 -7137.339,E2 -7137.339} C_VEL
LIN {X 0,Y 474.602,Z 70.863,A -85,B 0,C 180,E1 -7140.811,E2 -7140.811} C_VEL
LIN {X 0,Y 474.635,Z 70.848,A -85,B 0,C 180,E1 -7143.984,E2 -7143.984} C_VEL
LIN {X 0,Y 474.572,Z 70.866,A -85,B 0,C 180,E1 -7146.9,E2 -7146.9} C_VEL
LIN {X 0,Y 474.624,Z 70.86,A -85,B 0,C 180,E1 -7149.648,E2 -7149.648} C_VEL
LIN {X 0,Y 474.602,Z 70.845,A -85,B 0,C 180,E1 -7152.935,E2 -7152.935} C_VEL
LIN {X 0,Y 474.606,Z 70.866,A -85,B 0,C 180,E1 -7155.895,E2 -7155.895} C_VEL
LIN {X 0,Y 474.638,Z 70.859,A -85,B 0,C 180,E1 -7159.039,E2 -7159.039} C_VEL
LIN {X 0,Y 474.612,Z 70.865,A -85,B 0,C 180,E1 -7161.704,E2 -7161.704} C_VEL
LIN {X 0,Y 474.628,Z 70.859,A -85,B 0,C 180,E1 -7164.727,E2 -7164.727} C_VEL
LIN {X 0,Y 474.633,Z 70.86,A -85,B 0,C 180,E1 -7167.788,E2 -7167.788} C_VEL
LIN {X 0,Y 474.622,Z 70.863,A -85,B 0,C 180,E1 -7170.885,E2 -7170.885} C_VEL
LIN {X 0,Y 474.658,Z 70.85,A -85,B 0,C 180,E1 -7173.629,E2 -7173.629} C_VEL
LIN {X 0,Y 474.634,Z 70.864,A -85,B 0,C 180,E1 -7176.642,E2 -7176.642} C_VEL
LIN {X 0,Y 474.653,Z 70.85,A -85,B 0,C 180,E1 -7180.09,E2 -7180.09} C_VEL
LIN {X 0,Y 474.649,Z 70.857,A -85,B 0,C 180,E1 -7182.775,E2 -7182.775} C_VEL
LIN {X 0,Y 474.647,Z 70.857,A -85,B 0,C 180,E1 -7185.421,E2 -7185.421} C_VEL
LIN {X 0,Y 474.738,Z 70.846,A -85,B 0,C 180,E1 -7188.039,E2 -7188.039} C_VEL
LIN {X 0,Y 474.727,Z 70.837,A -85,B 0,C 180,E1 -7191.487,E2 -7191.487} C_VEL
LIN {X 0,Y 474.778,Z 70.844,A -85,B 0,C 180,E1 -7194.053,E2 -7194.053} C_VEL
LIN {X 0,Y 474.893,Z 70.824,A -85,B 0,C 180,E1 -7197.456,E2 -7197.456} C_VEL
LIN {X 0,Y 474.911,Z 70.814,A -85,B 0,C 180,E1 -7200,E2 -7200} C_VEL
LIN {X 0,Y 474.894,Z 70.825,A -85,B 0,C 180,E1 -7202.545,E2 -7202.545} C_VEL
LIN {X 0,Y 474.779,Z 70.844,A -85,B 0,C 180,E1 -7205.948,E2 -7205.948} C_VEL
LIN {X 0,Y 474.728,Z 70.836,A -85,B 0,C 180,E1 -7208.514,E2 -7208.514} C_VEL
LIN {X 0,Y 474.705,Z 70.85,A -85,B 0,C 180,E1 -7211.963,E2 -7211.963} C_VEL
LIN {X 0,Y 474.701,Z 70.855,A -85,B 0,C 180,E1 -7215.456,E2 -7215.456} C_VEL
LIN {X 0,Y 474.666,Z 70.843,A -85,B 0,C 180,E1 -7219.011,E2 -7219.011} C_VEL
LIN {X 0,Y 474.59,Z 70.866,A -85,B 0,C 180,E1 -7221.729,E2 -7221.729} C_VEL
LIN {X 0,Y 474.66,Z 70.854,A -85,B 0,C 180,E1 -7224.493,E2 -7224.493} C_VEL
LIN {X 0,Y 474.682,Z 70.848,A -85,B 0,C 180,E1 -7227.335,E2 -7227.335} C_VEL
LIN {X 0,Y 474.606,Z 70.862,A -85,B 0,C 180,E1 -7230.231,E2 -7230.231} C_VEL
LIN {X 0,Y 474.644,Z 70.853,A -85,B 0,C 180,E1 -7233.22,E2 -7233.22} C_VEL
LIN {X 0,Y 474.591,Z 70.864,A -85,B 0,C 180,E1 -7236.324,E2 -7236.324} C_VEL
LIN {X 0,Y 474.62,Z 70.855,A -85,B 0,C 180,E1 -7239.647,E2 -7239.647} C_VEL
LIN {X 0,Y 474.616,Z 70.865,A -85,B 0,C 180,E1 -7242.935,E2 -7242.935} C_VEL
LIN {X 0,Y 474.608,Z 70.862,A -85,B 0,C 180,E1 -7245.895,E2 -7245.895} C_VEL
LIN {X 0,Y 474.629,Z 70.851,A -85,B 0,C 180,E1 -7249.041,E2 -7249.041} C_VEL
LIN {X 0,Y 474.612,Z 70.861,A -85,B 0,C 180,E1 -7251.704,E2 -7251.704} C_VEL
LIN {X 0,Y 474.631,Z 70.856,A -85,B 0,C 180,E1 -7254.726,E2 -7254.726} C_VEL
LIN {X 0,Y 474.638,Z 70.859,A -85,B 0,C 180,E1 -7257.788,E2 -7257.788} C_VEL
LIN {X 0,Y 474.627,Z 70.863,A -85,B 0,C 180,E1 -7260.885,E2 -7260.885} C_VEL
LIN {X 0,Y 474.7,Z 70.934,A -85,B 0,C 180,E1 -7262.68,E2 -7262.68} C_VEL
LIN {X 0,Y 476.285,Z 79.94,A -85,B 0,C 180,E1 -7264.898,E2 -7264.898} C_VEL
LIN {X 0,Y 476.055,Z 88.095,A -85,B 0,C 180,E1 -7266.74,E2 -7266.74} C_VEL
LIN {X 0,Y 475.504,Z 102.584,A -85,B 0,C 180,E1 -7269.901,E2 -7269.901} C_VEL
LIN {X 0,Y 475.042,Z 113.882,A -85,B 0,C 180,E1 -7272.345,E2 -7272.345} C_VEL
LIN {X 0,Y 474.932,Z 117.833,A -85,B 0,C 180,E1 -7273.204,E2 -7273.204} C_VEL
LIN {X 0,Y 475.604,Z 122.014,A -85,B 0,C 180,E1 -7273.337,E2 -7273.337} C_VEL
LIN {X 0,Y 477.991,Z 137.391,A -85,B 0,C 180,E1 -7273.657,E2 -7273.657} C_VEL
LIN {X 0,Y 477.401,Z 222.715,A -85,B 0,C 180,E1 -7274.962,E2 -7274.962} C_VEL
LIN {X 0,Y 477.169,Z 232.611,A -85,B 0,C 180,E1 -7275.2,E2 -7275.2} C_VEL
LIN {X 0,Y 476.908,Z 242.59,A -85,B 0,C 180,E1 -7275.546,E2 -7275.546} C_VEL
LIN {X 0,Y 476.5,Z 252.953,A -85,B 0,C 180,E1 -7276.024,E2 -7276.024} C_VEL
LIN {X 0,Y 476.163,Z 262.093,A -85,B 0,C 180,E1 -7276.558,E2 -7276.558} C_VEL
LIN {X 0,Y 475.718,Z 271.087,A -85,B 0,C 180,E1 -7277.197,E2 -7277.197} C_VEL
LIN {X 0,Y 475.442,Z 278.957,A -85,B 0,C 180,E1 -7277.866,E2 -7277.866} C_VEL
LIN {X 0,Y 475.065,Z 287.216,A -85,B 0,C 180,E1 -7278.696,E2 -7278.696} C_VEL
LIN {X 0,Y 474.729,Z 294.437,A -85,B 0,C 180,E1 -7279.552,E2 -7279.552} C_VEL
LIN {X 0,Y 474.449,Z 300.639,A -85,B 0,C 180,E1 -7280.407,E2 -7280.407} C_VEL
LIN {X 0,Y 474.196,Z 307.176,A -85,B 0,C 180,E1 -7281.477,E2 -7281.477} C_VEL
LIN {X 0,Y 474.029,Z 311.677,A -85,B 0,C 180,E1 -7282.332,E2 -7282.332} C_VEL
LIN {X 0,Y 473.861,Z 317.003,A -85,B 0,C 180,E1 -7283.569,E2 -7283.569} C_VEL
LIN {X 0,Y 473.826,Z 321.489,A -85,B 0,C 180,E1 -7284.894,E2 -7284.894} C_VEL
LIN {X 0,Y 473.734,Z 323.852,A -85,B 0,C 180,E1 -7285.746,E2 -7285.746} C_VEL
LIN {X 0,Y 473.795,Z 325.65,A -85,B 0,C 180,E1 -7286.598,E2 -7286.598} C_VEL
LIN {X 0,Y 473.698,Z 328.088,A -85,B 0,C 180,E1 -7288.3,E2 -7288.3} C_VEL
LIN {X 0,Y 473.691,Z 328.675,A -85,B 0,C 180,E1 -7289.15,E2 -7289.15} C_VEL
LIN {X 0,Y 473.691,Z 328.675,A -85,B 0,C 180,E1 -7290.85,E2 -7290.85} C_VEL
LIN {X 0,Y 473.698,Z 328.088,A -85,B 0,C 180,E1 -7291.7,E2 -7291.7} C_VEL
LIN {X 0,Y 473.795,Z 325.65,A -85,B 0,C 180,E1 -7293.402,E2 -7293.402} C_VEL
LIN {X 0,Y 473.762,Z 322.703,A -85,B 0,C 180,E1 -7294.68,E2 -7294.68} C_VEL
LIN {X 0,Y 473.818,Z 318.719,A -85,B 0,C 180,E1 -7295.96,E2 -7295.96} C_VEL
LIN {X 0,Y 473.946,Z 313.592,A -85,B 0,C 180,E1 -7297.241,E2 -7297.241} C_VEL
LIN {X 0,Y 474.157,Z 308.332,A -85,B 0,C 180,E1 -7298.309,E2 -7298.309} C_VEL
LIN {X 0,Y 474.372,Z 302.014,A -85,B 0,C 180,E1 -7299.379,E2 -7299.379} C_VEL
LIN {X 0,Y 474.626,Z 296.063,A -85,B 0,C 180,E1 -7300.235,E2 -7300.235} C_VEL
LIN {X 0,Y 474.982,Z 289.136,A -85,B 0,C 180,E1 -7301.09,E2 -7301.09} C_VEL
LIN {X 0,Y 475.353,Z 280.955,A -85,B 0,C 180,E1 -7301.946,E2 -7301.946} C_VEL
LIN {X 0,Y 475.677,Z 273.042,A -85,B 0,C 180,E1 -7302.647,E2 -7302.647} C_VEL
LIN {X 0,Y 476.099,Z 263.727,A -85,B 0,C 180,E1 -7303.335,E2 -7303.335} C_VEL
LIN {X 0,Y 476.468,Z 253.96,A -85,B 0,C 180,E1 -7303.923,E2 -7303.923} C_VEL
LIN {X 0,Y 476.8,Z 245.165,A -85,B 0,C 180,E1 -7304.348,E2 -7304.348} C_VEL
LIN {X 0,Y 477.123,Z 235.235,A -85,B 0,C 180,E1 -7304.72,E2 -7304.72} C_VEL
LIN {X 0,Y 477.357,Z 225.378,A -85,B 0,C 180,E1 -7304.985,E2 -7304.985} C_VEL
LIN {X 0,Y 477.649,Z 199.685,A -85,B 0,C 180,E1 -7305.402,E2 -7305.402} C_VEL
LIN {X 0,Y 477.845,Z 135.159,A -85,B 0,C 180,E1 -7306.382,E2 -7306.382} C_VEL
LIN {X 0,Y 474.946,Z 118.259,A -85,B 0,C 180,E1 -7306.761,E2 -7306.761} C_VEL
LIN {X 0,Y 474.922,Z 117.113,A -85,B 0,C 180,E1 -7306.916,E2 -7306.916} C_VEL
LIN {X 0,Y 475.458,Z 103.824,A -85,B 0,C 180,E1 -7309.875,E2 -7309.875} C_VEL
LIN {X 0,Y 476.062,Z 88.185,A -85,B 0,C 180,E1 -7313.26,E2 -7313.26} C_VEL
LIN {X 0,Y 476.372,Z 80.963,A -85,B 0,C 180,E1 -7314.864,E2 -7314.864} C_VEL
LIN {X 0,Y 474.736,Z 71.073,A -85,B 0,C 180,E1 -7317.251,E2 -7317.251} C_VEL
LIN {X 0,Y 474.649,Z 70.862,A -85,B 0,C 180,E1 -7318.282,E2 -7318.282} C_VEL
LIN {X 0,Y 474.601,Z 70.868,A -85,B 0,C 180,E1 -7321.217,E2 -7321.217} C_VEL
LIN {X 0,Y 474.636,Z 70.859,A -85,B 0,C 180,E1 -7324.241,E2 -7324.241} C_VEL
LIN {X 0,Y 474.594,Z 70.868,A -85,B 0,C 180,E1 -7327.383,E2 -7327.383} C_VEL
LIN {X 0,Y 474.619,Z 70.851,A -85,B 0,C 180,E1 -7330.657,E2 -7330.657} C_VEL
LIN {X 0,Y 474.602,Z 70.87,A -85,B 0,C 180,E1 -7333.481,E2 -7333.481} C_VEL
LIN {X 0,Y 474.601,Z 70.863,A -85,B 0,C 180,E1 -7336.519,E2 -7336.519} C_VEL
LIN {X 0,Y 474.618,Z 70.861,A -85,B 0,C 180,E1 -7339.342,E2 -7339.342} C_VEL
LIN {X 0,Y 474.591,Z 70.866,A -85,B 0,C 180,E1 -7342.616,E2 -7342.616} C_VEL
LIN {X 0,Y 474.633,Z 70.851,A -85,B 0,C 180,E1 -7345.759,E2 -7345.759} C_VEL
LIN {X 0,Y 474.6,Z 70.867,A -85,B 0,C 180,E1 -7348.782,E2 -7348.782} C_VEL
LIN {X 0,Y 474.647,Z 70.851,A -85,B 0,C 180,E1 -7351.717,E2 -7351.717} C_VEL
LIN {X 0,Y 474.67,Z 70.851,A -85,B 0,C 180,E1 -7354.578,E2 -7354.578} C_VEL
LIN {X 0,Y 474.602,Z 70.862,A -85,B 0,C 180,E1 -7357.355,E2 -7357.355} C_VEL
LIN {X 0,Y 474.656,Z 70.851,A -85,B 0,C 180,E1 -7360.089,E2 -7360.089} C_VEL
LIN {X 0,Y 474.649,Z 70.856,A -85,B 0,C 180,E1 -7362.774,E2 -7362.774} C_VEL
LIN {X 0,Y 474.649,Z 70.856,A -85,B 0,C 180,E1 -7365.421,E2 -7365.421} C_VEL
LIN {X 0,Y 474.705,Z 70.85,A -85,B 0,C 180,E1 -7368.037,E2 -7368.037} C_VEL
LIN {X 0,Y 474.728,Z 70.836,A -85,B 0,C 180,E1 -7371.486,E2 -7371.486} C_VEL
LIN {X 0,Y 474.779,Z 70.844,A -85,B 0,C 180,E1 -7374.052,E2 -7374.052} C_VEL
LIN {X 0,Y 474.894,Z 70.825,A -85,B 0,C 180,E1 -7377.455,E2 -7377.455} C_VEL
LIN {X 0,Y 474.911,Z 70.814,A -85,B 0,C 180,E1 -7380,E2 -7380} C_VEL
LIN {X 0,Y 474.893,Z 70.824,A -85,B 0,C 180,E1 -7382.544,E2 -7382.544} C_VEL
LIN {X 0,Y 474.778,Z 70.844,A -85,B 0,C 180,E1 -7385.947,E2 -7385.947} C_VEL
LIN {X 0,Y 474.727,Z 70.837,A -85,B 0,C 180,E1 -7388.513,E2 -7388.513} C_VEL
LIN {X 0,Y 474.738,Z 70.846,A -85,B 0,C 180,E1 -7391.961,E2 -7391.961} C_VEL
LIN {X 0,Y 474.679,Z 70.854,A -85,B 0,C 180,E1 -7395.768,E2 -7395.768} C_VEL
LIN {X 0,Y 474.663,Z 70.846,A -85,B 0,C 180,E1 -7399.01,E2 -7399.01} C_VEL
LIN {X 0,Y 474.587,Z 70.866,A -85,B 0,C 180,E1 -7401.728,E2 -7401.728} C_VEL
LIN {X 0,Y 474.657,Z 70.856,A -85,B 0,C 180,E1 -7404.492,E2 -7404.492} C_VEL
LIN {X 0,Y 474.697,Z 70.846,A -85,B 0,C 180,E1 -7407.338,E2 -7407.338} C_VEL
LIN {X 0,Y 474.603,Z 70.868,A -85,B 0,C 180,E1 -7410.81,E2 -7410.81} C_VEL
LIN {X 0,Y 474.636,Z 70.852,A -85,B 0,C 180,E1 -7413.984,E2 -7413.984} C_VEL
LIN {X 0,Y 474.573,Z 70.873,A -85,B 0,C 180,E1 -7416.9,E2 -7416.9} C_VEL
LIN {X 0,Y 474.645,Z 70.854,A -85,B 0,C 180,E1 -7419.65,E2 -7419.65} C_VEL
LIN {X 0,Y 474.612,Z 70.865,A -85,B 0,C 180,E1 -7422.934,E2 -7422.934} C_VEL
LIN {X 0,Y 474.604,Z 70.859,A -85,B 0,C 180,E1 -7425.895,E2 -7425.895} C_VEL
LIN {X 0,Y 474.624,Z 70.851,A -85,B 0,C 180,E1 -7429.04,E2 -7429.04} C_VEL
LIN {X 0,Y 474.607,Z 70.864,A -85,B 0,C 180,E1 -7431.704,E2 -7431.704} C_VEL
LIN {X 0,Y 474.627,Z 70.848,A -85,B 0,C 180,E1 -7434.726,E2 -7434.726} C_VEL
LIN {X 0,Y 474.633,Z 70.862,A -85,B 0,C 180,E1 -7437.788,E2 -7437.788} C_VEL
LIN {X 0,Y 474.62,Z 70.853,A -85,B 0,C 180,E1 -7440.884,E2 -7440.884} C_VEL
LIN {X 0,Y 474.658,Z 70.862,A -85,B 0,C 180,E1 -7443.628,E2 -7443.628} C_VEL
LIN {X 0,Y 474.632,Z 70.861,A -85,B 0,C 180,E1 -7446.641,E2 -7446.641} C_VEL
LIN {X 0,Y 474.653,Z 70.861,A -85,B 0,C 180,E1 -7450.09,E2 -7450.09} C_VEL
LIN {X 0,Y 474.652,Z 70.863,A -85,B 0,C 180,E1 -7451.668,E2 -7451.668} C_VEL
LIN {X 0,Y 473.989,Z 70.946,A -85,B 0,C 180,E1 -7452.377,E2 -7452.377} C_VEL
LIN {X 0,Y 471.14,Z 71.303,A -85,B 0,C 180,E1 -7453.528,E2 -7453.528} C_VEL
LIN {X 0,Y 468.725,Z 71.603,A -85,B 0,C 180,E1 -7454.457,E2 -7454.457} C_VEL
LIN {X 0,Y 467.684,Z 71.73,A -85,B 0,C 180,E1 -7455.174,E2 -7455.174} C_VEL
LIN {X 0,Y 467.597,Z 71.74,A -85,B 0,C 180,E1 -7455.417,E2 -7455.417} C_VEL
LIN {X 0,Y 467.65,Z 71.733,A -85,B 0,C 180,E1 -7458.734,E2 -7458.734} C_VEL
LIN {X 0,Y 467.745,Z 71.721,A -85,B 0,C 180,E1 -7462.228,E2 -7462.228} C_VEL
LIN {X 0,Y 467.724,Z 71.726,A -85,B 0,C 180,E1 -7464.827,E2 -7464.827} C_VEL
LIN {X 0,Y 467.857,Z 71.71,A -85,B 0,C 180,E1 -7467.417,E2 -7467.417} C_VEL
LIN {X 0,Y 467.88,Z 71.704,A -85,B 0,C 180,E1 -7470,E2 -7470} C_VEL
LIN {X 0,Y 467.857,Z 71.709,A -85,B 0,C 180,E1 -7472.583,E2 -7472.583} C_VEL
LIN {X 0,Y 467.743,Z 71.721,A -85,B 0,C 180,E1 -7476.037,E2 -7476.037} C_VEL
LIN {X 0,Y 467.679,Z 71.732,A -85,B 0,C 180,E1 -7478.643,E2 -7478.643} C_VEL
LIN {X 0,Y 467.653,Z 71.734,A -85,B 0,C 180,E1 -7482.145,E2 -7482.145} C_VEL
LIN {X 0,Y 467.636,Z 71.734,A -85,B 0,C 180,E1 -7485.695,E2 -7485.695} C_VEL
LIN {X 0,Y 467.614,Z 71.739,A -85,B 0,C 180,E1 -7488.765,E2 -7488.765} C_VEL
LIN {X 0,Y 467.577,Z 71.74,A -85,B 0,C 180,E1 -7491.269,E2 -7491.269} C_VEL
LIN {X 0,Y 467.57,Z 71.745,A -85,B 0,C 180,E1 -7493.943,E2 -7493.943} C_VEL
LIN {X 0,Y 467.613,Z 71.736,A -85,B 0,C 180,E1 -7496.8,E2 -7496.8} C_VEL
LIN {X 0,Y 467.551,Z 71.735,A -85,B 0,C 180,E1 -7499.738,E2 -7499.738} C_VEL
LIN {X 0,Y 467.58,Z 71.736,A -85,B 0,C 180,E1 -7502.758,E2 -7502.758} C_VEL
LIN {X 0,Y 467.553,Z 71.735,A -85,B 0,C 180,E1 -7505.889,E2 -7505.889} C_VEL
LIN {X 0,Y 467.579,Z 71.74,A -85,B 0,C 180,E1 -7509.145,E2 -7509.145} C_VEL
LIN {X 0,Y 467.583,Z 71.717,A -85,B 0,C 180,E1 -7512.567,E2 -7512.567} C_VEL
LIN {X 0,Y 467.567,Z 71.736,A -85,B 0,C 180,E1 -7515.053,E2 -7515.053} C_VEL
LIN {X 0,Y 467.585,Z 71.742,A -85,B 0,C 180,E1 -7517.44,E2 -7517.44} C_VEL
LIN {X 0,Y 467.594,Z 71.735,A -85,B 0,C 180,E1 -7520.857,E2 -7520.857} C_VEL
LIN {X 0,Y 467.56,Z 71.737,A -85,B 0,C 180,E1 -7524.261,E2 -7524.261} C_VEL
LIN {X 0,Y 467.579,Z 71.743,A -85,B 0,C 180,E1 -7527.321,E2 -7527.321} C_VEL
LIN {X 0,Y 467.568,Z 71.742,A -85,B 0,C 180,E1 -7530.668,E2 -7530.668} C_VEL
LIN {X 0,Y 467.614,Z 71.729,A -85,B 0,C 180,E1 -7533.2,E2 -7533.2} C_VEL
LIN {X 0,Y 467.591,Z 71.739,A -85,B 0,C 180,E1 -7536.469,E2 -7536.469} C_VEL
LIN {X 0,Y 467.621,Z 71.725,A -85,B 0,C 180,E1 -7539.778,E2 -7539.778} C_VEL
LIN {X 0,Y 467.608,Z 71.729,A -85,B 0,C 180,E1 -7542.507,E2 -7542.507} C_VEL
LIN {X 0,Y 467.605,Z 71.735,A -85,B 0,C 180,E1 -7545.197,E2 -7545.197} C_VEL
LIN {X 0,Y 467.682,Z 71.723,A -85,B 0,C 180,E1 -7547.856,E2 -7547.856} C_VEL
LIN {X 0,Y 467.681,Z 71.714,A -85,B 0,C 180,E1 -7551.358,E2 -7551.358} C_VEL
LIN {X 0,Y 467.743,Z 71.719,A -85,B 0,C 180,E1 -7553.963,E2 -7553.963} C_VEL
LIN {X 0,Y 467.859,Z 71.7,A -85,B 0,C 180,E1 -7557.418,E2 -7557.418} C_VEL
LIN {X 0,Y 467.882,Z 71.688,A -85,B 0,C 180,E1 -7560,E2 -7560} C_VEL
LIN {X 0,Y 467.859,Z 71.701,A -85,B 0,C 180,E1 -7562.583,E2 -7562.583} C_VEL
LIN {X 0,Y 467.744,Z 71.719,A -85,B 0,C 180,E1 -7566.038,E2 -7566.038} C_VEL
LIN {X 0,Y 467.682,Z 71.713,A -85,B 0,C 180,E1 -7568.643,E2 -7568.643} C_VEL
LIN {X 0,Y 467.656,Z 71.726,A -85,B 0,C 180,E1 -7572.146,E2 -7572.146} C_VEL
LIN {X 0,Y 467.64,Z 71.731,A -85,B 0,C 180,E1 -7575.695,E2 -7575.695} C_VEL
LIN {X 0,Y 467.618,Z 71.719,A -85,B 0,C 180,E1 -7578.765,E2 -7578.765} C_VEL
LIN {X 0,Y 467.581,Z 71.737,A -85,B 0,C 180,E1 -7581.269,E2 -7581.269} C_VEL
LIN {X 0,Y 467.574,Z 71.737,A -85,B 0,C 180,E1 -7583.944,E2 -7583.944} C_VEL
LIN {X 0,Y 467.617,Z 71.726,A -85,B 0,C 180,E1 -7586.801,E2 -7586.801} C_VEL
LIN {X 0,Y 467.555,Z 71.741,A -85,B 0,C 180,E1 -7589.739,E2 -7589.739} C_VEL
LIN {X 0,Y 467.584,Z 71.74,A -85,B 0,C 180,E1 -7592.759,E2 -7592.759} C_VEL
LIN {X 0,Y 467.555,Z 71.738,A -85,B 0,C 180,E1 -7595.89,E2 -7595.89} C_VEL
LIN {X 0,Y 467.562,Z 71.737,A -85,B 0,C 180,E1 -7599.147,E2 -7599.147} C_VEL
LIN {X 0,Y 467.588,Z 71.743,A -85,B 0,C 180,E1 -7602.567,E2 -7602.567} C_VEL
LIN {X 0,Y 467.567,Z 71.74,A -85,B 0,C 180,E1 -7605.053,E2 -7605.053} C_VEL
LIN {X 0,Y 467.591,Z 71.736,A -85,B 0,C 180,E1 -7607.44,E2 -7607.44} C_VEL
LIN {X 0,Y 467.578,Z 71.737,A -85,B 0,C 180,E1 -7610.855,E2 -7610.855} C_VEL
LIN {X 0,Y 467.565,Z 71.737,A -85,B 0,C 180,E1 -7614.261,E2 -7614.261} C_VEL
LIN {X 0,Y 467.584,Z 71.738,A -85,B 0,C 180,E1 -7617.321,E2 -7617.321} C_VEL
LIN {X 0,Y 467.573,Z 71.74,A -85,B 0,C 180,E1 -7620.668,E2 -7620.668} C_VEL
LIN {X 0,Y 467.655,Z 71.784,A -85,B 0,C 180,E1 -7622.458,E2 -7622.458} C_VEL
LIN {X 0,Y 469.289,Z 80.827,A -85,B 0,C 180,E1 -7624.735,E2 -7624.735} C_VEL
LIN {X 0,Y 469.181,Z 87.93,A -85,B 0,C 180,E1 -7626.378,E2 -7626.378} C_VEL
LIN {X 0,Y 468.499,Z 103.455,A -85,B 0,C 180,E1 -7629.817,E2 -7629.817} C_VEL
LIN {X 0,Y 467.962,Z 115.642,A -85,B 0,C 180,E1 -7632.52,E2 -7632.52} C_VEL
LIN {X 0,Y 467.897,Z 117.622,A -85,B 0,C 180,E1 -7632.94,E2 -7632.94} C_VEL
LIN {X 0,Y 468.416,Z 120.83,A -85,B 0,C 180,E1 -7633.058,E2 -7633.058} C_VEL
LIN {X 0,Y 471.183,Z 137.91,A -85,B 0,C 180,E1 -7633.425,E2 -7633.425} C_VEL
LIN {X 0,Y 470.568,Z 222.525,A -85,B 0,C 180,E1 -7634.738,E2 -7634.738} C_VEL
LIN {X 0,Y 470.308,Z 232.421,A -85,B 0,C 180,E1 -7634.979,E2 -7634.979} C_VEL
LIN {X 0,Y 470.023,Z 242.399,A -85,B 0,C 180,E1 -7635.33,E2 -7635.33} C_VEL
LIN {X 0,Y 469.599,Z 252.762,A -85,B 0,C 180,E1 -7635.814,E2 -7635.814} C_VEL
LIN {X 0,Y 469.231,Z 261.898,A -85,B 0,C 180,E1 -7636.355,E2 -7636.355} C_VEL
LIN {X 0,Y 468.763,Z 270.896,A -85,B 0,C 180,E1 -7637.004,E2 -7637.004} C_VEL
LIN {X 0,Y 468.452,Z 278.969,A -85,B 0,C 180,E1 -7637.702,E2 -7637.702} C_VEL
LIN {X 0,Y 468.072,Z 287.025,A -85,B 0,C 180,E1 -7638.525,E2 -7638.525} C_VEL
LIN {X 0,Y 467.726,Z 294.245,A -85,B 0,C 180,E1 -7639.393,E2 -7639.393} C_VEL
LIN {X 0,Y 467.437,Z 300.448,A -85,B 0,C 180,E1 -7640.262,E2 -7640.262} C_VEL
LIN {X 0,Y 467.154,Z 306.985,A -85,B 0,C 180,E1 -7641.347,E2 -7641.347} C_VEL
LIN {X 0,Y 466.976,Z 311.486,A -85,B 0,C 180,E1 -7642.215,E2 -7642.215} C_VEL
LIN {X 0,Y 466.789,Z 317.161,A -85,B 0,C 180,E1 -7643.568,E2 -7643.568} C_VEL
LIN {X 0,Y 466.734,Z 321.298,A -85,B 0,C 180,E1 -7644.816,E2 -7644.816} C_VEL
LIN {X 0,Y 466.647,Z 323.661,A -85,B 0,C 180,E1 -7645.681,E2 -7645.681} C_VEL
LIN {X 0,Y 466.689,Z 325.459,A -85,B 0,C 180,E1 -7646.547,E2 -7646.547} C_VEL
LIN {X 0,Y 466.608,Z 327.898,A -85,B 0,C 180,E1 -7648.274,E2 -7648.274} C_VEL
LIN {X 0,Y 466.621,Z 328.485,A -85,B 0,C 180,E1 -7649.137,E2 -7649.137} C_VEL
LIN {X 0,Y 466.621,Z 328.485,A -85,B 0,C 180,E1 -7650.863,E2 -7650.863} C_VEL
LIN {X 0,Y 466.608,Z 327.898,A -85,B 0,C 180,E1 -7651.726,E2 -7651.726} C_VEL
LIN {X 0,Y 466.689,Z 325.459,A -85,B 0,C 180,E1 -7653.453,E2 -7653.453} C_VEL
LIN {X 0,Y 466.689,Z 322.513,A -85,B 0,C 180,E1 -7654.751,E2 -7654.751} C_VEL
LIN {X 0,Y 466.737,Z 318.528,A -85,B 0,C 180,E1 -7656.05,E2 -7656.05} C_VEL
LIN {X 0,Y 466.867,Z 313.4,A -85,B 0,C 180,E1 -7657.351,E2 -7657.351} C_VEL
LIN {X 0,Y 467.106,Z 308.141,A -85,B 0,C 180,E1 -7658.436,E2 -7658.436} C_VEL
LIN {X 0,Y 467.348,Z 301.823,A -85,B 0,C 180,E1 -7659.522,E2 -7659.522} C_VEL
LIN {X 0,Y 467.603,Z 295.871,A -85,B 0,C 180,E1 -7660.391,E2 -7660.391} C_VEL
LIN {X 0,Y 467.97,Z 288.944,A -85,B 0,C 180,E1 -7661.258,E2 -7661.258} C_VEL
LIN {X 0,Y 468.367,Z 280.763,A -85,B 0,C 180,E1 -7662.127,E2 -7662.127} C_VEL
LIN {X 0,Y 468.737,Z 272.851,A -85,B 0,C 180,E1 -7662.838,E2 -7662.838} C_VEL
LIN {X 0,Y 469.172,Z 263.531,A -85,B 0,C 180,E1 -7663.536,E2 -7663.536} C_VEL
LIN {X 0,Y 469.569,Z 253.77,A -85,B 0,C 180,E1 -7664.131,E2 -7664.131} C_VEL
LIN {X 0,Y 469.917,Z 244.974,A -85,B 0,C 180,E1 -7664.563,E2 -7664.563} C_VEL
LIN {X 0,Y 470.261,Z 235.045,A -85,B 0,C 180,E1 -7664.939,E2 -7664.939} C_VEL
LIN {X 0,Y 470.523,Z 225.188,A -85,B 0,C 180,E1 -7665.208,E2 -7665.208} C_VEL
LIN {X 0,Y 470.82,Z 199.655,A -85,B 0,C 180,E1 -7665.628,E2 -7665.628} C_VEL
LIN {X 0,Y 471.027,Z 135.967,A -85,B 0,C 180,E1 -7666.61,E2 -7666.61} C_VEL
LIN {X 0,Y 467.943,Z 118.001,A -85,B 0,C 180,E1 -7667.023,E2 -7667.023} C_VEL
LIN {X 0,Y 467.912,Z 116.501,A -85,B 0,C 180,E1 -7667.279,E2 -7667.279} C_VEL
LIN {X 0,Y 468.52,Z 103.665,A -85,B 0,C 180,E1 -7670.182,E2 -7670.182} C_VEL
LIN {X 0,Y 469.232,Z 87.006,A -85,B 0,C 180,E1 -7673.853,E2 -7673.853} C_VEL
LIN {X 0,Y 469.273,Z 80.826,A -85,B 0,C 180,E1 -7675.266,E2 -7675.266} C_VEL
LIN {X 0,Y 467.656,Z 71.767,A -85,B 0,C 180,E1 -7677.543,E2 -7677.543} C_VEL
LIN {X 0,Y 467.571,Z 71.743,A -85,B 0,C 180,E1 -7681.045,E2 -7681.045} C_VEL
LIN {X 0,Y 467.592,Z 71.737,A -85,B 0,C 180,E1 -7684.242,E2 -7684.242} C_VEL
LIN {X 0,Y 467.552,Z 71.743,A -85,B 0,C 180,E1 -7687.186,E2 -7687.186} C_VEL
LIN {X 0,Y 467.576,Z 71.729,A -85,B 0,C 180,E1 -7690.265,E2 -7690.265} C_VEL
LIN {X 0,Y 467.588,Z 71.737,A -85,B 0,C 180,E1 -7692.567,E2 -7692.567} C_VEL
LIN {X 0,Y 467.567,Z 71.741,A -85,B 0,C 180,E1 -7695.052,E2 -7695.052} C_VEL
LIN {X 0,Y 467.591,Z 71.743,A -85,B 0,C 180,E1 -7697.44,E2 -7697.44} C_VEL
LIN {X 0,Y 467.562,Z 71.737,A -85,B 0,C 180,E1 -7700.853,E2 -7700.853} C_VEL
LIN {X 0,Y 467.562,Z 71.738,A -85,B 0,C 180,E1 -7704.26,E2 -7704.26} C_VEL
LIN {X 0,Y 467.583,Z 71.74,A -85,B 0,C 180,E1 -7707.321,E2 -7707.321} C_VEL
LIN {X 0,Y 467.571,Z 71.743,A -85,B 0,C 180,E1 -7710.667,E2 -7710.667} C_VEL
LIN {X 0,Y 467.617,Z 71.726,A -85,B 0,C 180,E1 -7713.199,E2 -7713.199} C_VEL
LIN {X 0,Y 467.594,Z 71.738,A -85,B 0,C 180,E1 -7716.468,E2 -7716.468} C_VEL
LIN {X 0,Y 467.624,Z 71.725,A -85,B 0,C 180,E1 -7719.777,E2 -7719.777} C_VEL
LIN {X 0,Y 467.608,Z 71.727,A -85,B 0,C 180,E1 -7722.506,E2 -7722.506} C_VEL
LIN {X 0,Y 467.607,Z 71.733,A -85,B 0,C 180,E1 -7725.196,E2 -7725.196} C_VEL
LIN {X 0,Y 467.656,Z 71.726,A -85,B 0,C 180,E1 -7727.854,E2 -7727.854} C_VEL
LIN {X 0,Y 467.682,Z 71.713,A -85,B 0,C 180,E1 -7731.357,E2 -7731.357} C_VEL
LIN {X 0,Y 467.744,Z 71.719,A -85,B 0,C 180,E1 -7733.962,E2 -7733.962} C_VEL
LIN {X 0,Y 467.859,Z 71.701,A -85,B 0,C 180,E1 -7737.417,E2 -7737.417} C_VEL
LIN {X 0,Y 467.882,Z 71.688,A -85,B 0,C 180,E1 -7740,E2 -7740} C_VEL
LIN {X 0,Y 467.859,Z 71.7,A -85,B 0,C 180,E1 -7742.582,E2 -7742.582} C_VEL
LIN {X 0,Y 467.743,Z 71.719,A -85,B 0,C 180,E1 -7746.037,E2 -7746.037} C_VEL
LIN {X 0,Y 467.681,Z 71.714,A -85,B 0,C 180,E1 -7748.642,E2 -7748.642} C_VEL
LIN {X 0,Y 467.682,Z 71.723,A -85,B 0,C 180,E1 -7752.144,E2 -7752.144} C_VEL
LIN {X 0,Y 467.648,Z 71.729,A -85,B 0,C 180,E1 -7755.885,E2 -7755.885} C_VEL
LIN {X 0,Y 467.622,Z 71.724,A -85,B 0,C 180,E1 -7759.307,E2 -7759.307} C_VEL
LIN {X 0,Y 467.533,Z 71.743,A -85,B 0,C 180,E1 -7762.073,E2 -7762.073} C_VEL
LIN {X 0,Y 467.602,Z 71.739,A -85,B 0,C 180,E1 -7764.887,E2 -7764.887} C_VEL
LIN {X 0,Y 467.625,Z 71.724,A -85,B 0,C 180,E1 -7767.768,E2 -7767.768} C_VEL
LIN {X 0,Y 467.567,Z 71.746,A -85,B 0,C 180,E1 -7771.045,E2 -7771.045} C_VEL
LIN {X 0,Y 467.587,Z 71.731,A -85,B 0,C 180,E1 -7774.242,E2 -7774.242} C_VEL
LIN {X 0,Y 467.548,Z 71.745,A -85,B 0,C 180,E1 -7777.186,E2 -7777.186} C_VEL
LIN {X 0,Y 467.591,Z 71.736,A -85,B 0,C 180,E1 -7780.262,E2 -7780.262} C_VEL
LIN {X 0,Y 467.583,Z 71.742,A -85,B 0,C 180,E1 -7782.567,E2 -7782.567} C_VEL
LIN {X 0,Y 467.567,Z 71.735,A -85,B 0,C 180,E1 -7785.053,E2 -7785.053} C_VEL
LIN {X 0,Y 467.585,Z 71.717,A -85,B 0,C 180,E1 -7787.44,E2 -7787.44} C_VEL
LIN {X 0,Y 467.579,Z 71.74,A -85,B 0,C 180,E1 -7790.855,E2 -7790.855} C_VEL
LIN {X 0,Y 467.56,Z 71.733,A -85,B 0,C 180,E1 -7794.26,E2 -7794.26} C_VEL
LIN {X 0,Y 467.578,Z 71.737,A -85,B 0,C 180,E1 -7797.321,E2 -7797.321} C_VEL
LIN {X 0,Y 467.566,Z 71.731,A -85,B 0,C 180,E1 -7800.667,E2 -7800.667} C_VEL
LIN {X 0,Y 467.613,Z 71.736,A -85,B 0,C 180,E1 -7803.2,E2 -7803.2} C_VEL
LIN {X 0,Y 467.59,Z 71.739,A -85,B 0,C 180,E1 -7806.468,E2 -7806.468} C_VEL
LIN {X 0,Y 467.621,Z 71.739,A -85,B 0,C 180,E1 -7809.777,E2 -7809.777} C_VEL
LIN {X 0,Y 467.606,Z 71.737,A -85,B 0,C 180,E1 -7812.507,E2 -7812.507} C_VEL
LIN {X 0,Y 467.597,Z 71.74,A -85,B 0,C 180,E1 -7815.417,E2 -7815.417} C_VEL
LIN {X 0,Y 466.926,Z 71.823,A -85,B 0,C 180,E1 -7816.136,E2 -7816.136} C_VEL
LIN {X 0,Y 464.081,Z 72.18,A -85,B 0,C 180,E1 -7817.304,E2 -7817.304} C_VEL
LIN {X 0,Y 461.682,Z 72.476,A -85,B 0,C 180,E1 -7818.246,E2 -7818.246} C_VEL
LIN {X 0,Y 460.656,Z 72.606,A -85,B 0,C 180,E1 -7818.974,E2 -7818.974} C_VEL
LIN {X 0,Y 460.574,Z 72.615,A -85,B 0,C 180,E1 -7819.22,E2 -7819.22} C_VEL
LIN {X 0,Y 460.716,Z 72.597,A -85,B 0,C 180,E1 -7822.538,E2 -7822.538} C_VEL
LIN {X 0,Y 460.696,Z 72.601,A -85,B 0,C 180,E1 -7824.748,E2 -7824.748} C_VEL
LIN {X 0,Y 460.822,Z 72.586,A -85,B 0,C 180,E1 -7827.378,E2 -7827.378} C_VEL
LIN {X 0,Y 460.85,Z 72.58,A -85,B 0,C 180,E1 -7830,E2 -7830} C_VEL
LIN {X 0,Y 460.822,Z 72.586,A -85,B 0,C 180,E1 -7832.622,E2 -7832.622} C_VEL
LIN {X 0,Y 460.708,Z 72.598,A -85,B 0,C 180,E1 -7836.13,E2 -7836.13} C_VEL
LIN {X 0,Y 460.626,Z 72.611,A -85,B 0,C 180,E1 -7838.776,E2 -7838.776} C_VEL
LIN {X 0,Y 460.61,Z 72.612,A -85,B 0,C 180,E1 -7842.445,E2 -7842.445} C_VEL
LIN {X 0,Y 460.596,Z 72.613,A -85,B 0,C 180,E1 -7845.998,E2 -7845.998} C_VEL
LIN {X 0,Y 460.568,Z 72.616,A -85,B 0,C 180,E1 -7848.902,E2 -7848.902} C_VEL
LIN {X 0,Y 460.513,Z 72.621,A -85,B 0,C 180,E1 -7851.486,E2 -7851.486} C_VEL
LIN {X 0,Y 460.539,Z 72.621,A -85,B 0,C 180,E1 -7854.332,E2 -7854.332} C_VEL
LIN {X 0,Y 460.576,Z 72.612,A -85,B 0,C 180,E1 -7857.244,E2 -7857.244} C_VEL
LIN {X 0,Y 460.508,Z 72.618,A -85,B 0,C 180,E1 -7860.24,E2 -7860.24} C_VEL
LIN {X 0,Y 460.526,Z 72.616,A -85,B 0,C 180,E1 -7863.325,E2 -7863.325} C_VEL
LIN {X 0,Y 460.476,Z 72.622,A -85,B 0,C 180,E1 -7866.529,E2 -7866.529} C_VEL
LIN {X 0,Y 460.542,Z 72.615,A -85,B 0,C 180,E1 -7868.898,E2 -7868.898} C_VEL
LIN {X 0,Y 460.519,Z 72.596,A -85,B 0,C 180,E1 -7872.182,E2 -7872.182} C_VEL
LIN {X 0,Y 460.513,Z 72.619,A -85,B 0,C 180,E1 -7875.412,E2 -7875.412} C_VEL
LIN {X 0,Y 460.532,Z 72.612,A -85,B 0,C 180,E1 -7878.397,E2 -7878.397} C_VEL
LIN {X 0,Y 460.535,Z 72.619,A -85,B 0,C 180,E1 -7881.269,E2 -7881.269} C_VEL
LIN {X 0,Y 460.511,Z 72.616,A -85,B 0,C 180,E1 -7884.555,E2 -7884.555} C_VEL
LIN {X 0,Y 460.529,Z 72.617,A -85,B 0,C 180,E1 -7887.716,E2 -7887.716} C_VEL
LIN {X 0,Y 460.538,Z 72.619,A -85,B 0,C 180,E1 -7890.77,E2 -7890.77} C_VEL
LIN {X 0,Y 460.561,Z 72.605,A -85,B 0,C 180,E1 -7893.735,E2 -7893.735} C_VEL
LIN {X 0,Y 460.544,Z 72.619,A -85,B 0,C 180,E1 -7896.624,E2 -7896.624} C_VEL
LIN {X 0,Y 460.549,Z 72.606,A -85,B 0,C 180,E1 -7899.453,E2 -7899.453} C_VEL
LIN {X 0,Y 460.558,Z 72.603,A -85,B 0,C 180,E1 -7902.231,E2 -7902.231} C_VEL
LIN {X 0,Y 460.564,Z 72.614,A -85,B 0,C 180,E1 -7904.965,E2 -7904.965} C_VEL
LIN {X 0,Y 460.629,Z 72.6,A -85,B 0,C 180,E1 -7907.667,E2 -7907.667} C_VEL
LIN {X 0,Y 460.628,Z 72.592,A -85,B 0,C 180,E1 -7911.224,E2 -7911.224} C_VEL
LIN {X 0,Y 460.709,Z 72.594,A -85,B 0,C 180,E1 -7913.871,E2 -7913.871} C_VEL
LIN {X 0,Y 460.8,Z 72.579,A -85,B 0,C 180,E1 -7917.378,E2 -7917.378} C_VEL
LIN {X 0,Y 460.852,Z 72.563,A -85,B 0,C 180,E1 -7920,E2 -7920} C_VEL
LIN {X 0,Y 460.8,Z 72.58,A -85,B 0,C 180,E1 -7922.623,E2 -7922.623} C_VEL
LIN {X 0,Y 460.71,Z 72.594,A -85,B 0,C 180,E1 -7926.13,E2 -7926.13} C_VEL
LIN {X 0,Y 460.629,Z 72.591,A -85,B 0,C 180,E1 -7928.777,E2 -7928.777} C_VEL
LIN {X 0,Y 460.614,Z 72.602,A -85,B 0,C 180,E1 -7932.445,E2 -7932.445} C_VEL
LIN {X 0,Y 460.601,Z 72.604,A -85,B 0,C 180,E1 -7935.998,E2 -7935.998} C_VEL
LIN {X 0,Y 460.571,Z 72.597,A -85,B 0,C 180,E1 -7938.902,E2 -7938.902} C_VEL
LIN {X 0,Y 460.517,Z 72.621,A -85,B 0,C 180,E1 -7941.486,E2 -7941.486} C_VEL
LIN {X 0,Y 460.544,Z 72.612,A -85,B 0,C 180,E1 -7944.333,E2 -7944.333} C_VEL
LIN {X 0,Y 460.574,Z 72.603,A -85,B 0,C 180,E1 -7947.244,E2 -7947.244} C_VEL
LIN {X 0,Y 460.512,Z 72.618,A -85,B 0,C 180,E1 -7950.24,E2 -7950.24} C_VEL
LIN {X 0,Y 460.53,Z 72.609,A -85,B 0,C 180,E1 -7953.325,E2 -7953.325} C_VEL
LIN {X 0,Y 460.478,Z 72.624,A -85,B 0,C 180,E1 -7956.53,E2 -7956.53} C_VEL
LIN {X 0,Y 460.527,Z 72.611,A -85,B 0,C 180,E1 -7959.863,E2 -7959.863} C_VEL
LIN {X 0,Y 460.514,Z 72.622,A -85,B 0,C 180,E1 -7962.901,E2 -7962.901} C_VEL
LIN {X 0,Y 460.51,Z 72.618,A -85,B 0,C 180,E1 -7965.831,E2 -7965.831} C_VEL
LIN {X 0,Y 460.532,Z 72.606,A -85,B 0,C 180,E1 -7968.989,E2 -7968.989} C_VEL
LIN {X 0,Y 460.525,Z 72.615,A -85,B 0,C 180,E1 -7971.267,E2 -7971.267} C_VEL
LIN {X 0,Y 460.515,Z 72.614,A -85,B 0,C 180,E1 -7974.555,E2 -7974.555} C_VEL
LIN {X 0,Y 460.534,Z 72.616,A -85,B 0,C 180,E1 -7977.716,E2 -7977.716} C_VEL
LIN {X 0,Y 460.543,Z 72.616,A -85,B 0,C 180,E1 -7980.769,E2 -7980.769} C_VEL
LIN {X 0,Y 460.621,Z 72.663,A -85,B 0,C 180,E1 -7982.245,E2 -7982.245} C_VEL
LIN {X 0,Y 462.416,Z 82.736,A -85,B 0,C 180,E1 -7984.814,E2 -7984.814} C_VEL
LIN {X 0,Y 461.989,Z 92.944,A -85,B 0,C 180,E1 -7987.175,E2 -7987.175} C_VEL
LIN {X 0,Y 461.403,Z 106.393,A -85,B 0,C 180,E1 -7990.19,E2 -7990.19} C_VEL
LIN {X 0,Y 460.876,Z 117.436,A -85,B 0,C 180,E1 -7992.672,E2 -7992.672} C_VEL
LIN {X 0,Y 461.393,Z 120.398,A -85,B 0,C 180,E1 -7992.789,E2 -7992.789} C_VEL
LIN {X 0,Y 464.326,Z 137.718,A -85,B 0,C 180,E1 -7993.173,E2 -7993.173} C_VEL
LIN {X 0,Y 463.713,Z 222.334,A -85,B 0,C 180,E1 -7994.507,E2 -7994.507} C_VEL
LIN {X 0,Y 463.461,Z 232.231,A -85,B 0,C 180,E1 -7994.752,E2 -7994.752} C_VEL
LIN {X 0,Y 463.159,Z 242.208,A -85,B 0,C 180,E1 -7995.107,E2 -7995.107} C_VEL
LIN {X 0,Y 462.724,Z 252.572,A -85,B 0,C 180,E1 -7995.599,E2 -7995.599} C_VEL
LIN {X 0,Y 462.325,Z 261.708,A -85,B 0,C 180,E1 -7996.148,E2 -7996.148} C_VEL
LIN {X 0,Y 461.832,Z 270.705,A -85,B 0,C 180,E1 -7996.805,E2 -7996.805} C_VEL
LIN {X 0,Y 461.467,Z 278.97,A -85,B 0,C 180,E1 -7997.532,E2 -7997.532} C_VEL
LIN {X 0,Y 461.086,Z 286.833,A -85,B 0,C 180,E1 -7998.348,E2 -7998.348} C_VEL
LIN {X 0,Y 460.715,Z 294.054,A -85,B 0,C 180,E1 -7999.23,E2 -7999.23} C_VEL
LIN {X 0,Y 460.399,Z 300.256,A -85,B 0,C 180,E1 -8000.112,E2 -8000.112} C_VEL
LIN {X 0,Y 460.113,Z 306.794,A -85,B 0,C 180,E1 -8001.214,E2 -8001.214} C_VEL
LIN {X 0,Y 459.898,Z 311.294,A -85,B 0,C 180,E1 -8002.095,E2 -8002.095} C_VEL
LIN {X 0,Y 459.736,Z 316.277,A -85,B 0,C 180,E1 -8003.273,E2 -8003.273} C_VEL
LIN {X 0,Y 459.646,Z 321.107,A -85,B 0,C 180,E1 -8004.736,E2 -8004.736} C_VEL
LIN {X 0,Y 459.564,Z 323.47,A -85,B 0,C 180,E1 -8005.615,E2 -8005.615} C_VEL
LIN {X 0,Y 459.584,Z 325.268,A -85,B 0,C 180,E1 -8006.493,E2 -8006.493} C_VEL
LIN {X 0,Y 459.521,Z 327.707,A -85,B 0,C 180,E1 -8008.247,E2 -8008.247} C_VEL
LIN {X 0,Y 459.524,Z 328.295,A -85,B 0,C 180,E1 -8009.124,E2 -8009.124} C_VEL
LIN {X 0,Y 459.524,Z 328.295,A -85,B 0,C 180,E1 -8010.876,E2 -8010.876} C_VEL
LIN {X 0,Y 459.521,Z 327.707,A -85,B 0,C 180,E1 -8011.753,E2 -8011.753} C_VEL
LIN {X 0,Y 459.584,Z 325.268,A -85,B 0,C 180,E1 -8013.507,E2 -8013.507} C_VEL
LIN {X 0,Y 459.617,Z 322.323,A -85,B 0,C 180,E1 -8014.824,E2 -8014.824} C_VEL
LIN {X 0,Y 459.648,Z 318.337,A -85,B 0,C 180,E1 -8016.144,E2 -8016.144} C_VEL
LIN {X 0,Y 459.813,Z 313.209,A -85,B 0,C 180,E1 -8017.465,E2 -8017.465} C_VEL
LIN {X 0,Y 460.042,Z 307.949,A -85,B 0,C 180,E1 -8018.566,E2 -8018.566} C_VEL
LIN {X 0,Y 460.318,Z 301.632,A -85,B 0,C 180,E1 -8019.668,E2 -8019.668} C_VEL
LIN {X 0,Y 460.588,Z 295.68,A -85,B 0,C 180,E1 -8020.551,E2 -8020.551} C_VEL
LIN {X 0,Y 460.979,Z 288.753,A -85,B 0,C 180,E1 -8021.431,E2 -8021.431} C_VEL
LIN {X 0,Y 461.394,Z 280.572,A -85,B 0,C 180,E1 -8022.313,E2 -8022.313} C_VEL
LIN {X 0,Y 461.827,Z 271.763,A -85,B 0,C 180,E1 -8023.108,E2 -8023.108} C_VEL
LIN {X 0,Y 462.239,Z 263.34,A -85,B 0,C 180,E1 -8023.743,E2 -8023.743} C_VEL
LIN {X 0,Y 462.663,Z 253.579,A -85,B 0,C 180,E1 -8024.347,E2 -8024.347} C_VEL
LIN {X 0,Y 463.13,Z 243.497,A -85,B 0,C 180,E1 -8024.837,E2 -8024.837} C_VEL
LIN {X 0,Y 463.448,Z 233.98,A -85,B 0,C 180,E1 -8025.192,E2 -8025.192} C_VEL
LIN {X 0,Y 463.708,Z 223.666,A -85,B 0,C 180,E1 -8025.465,E2 -8025.465} C_VEL
LIN {X 0,Y 464.303,Z 147.202,A -85,B 0,C 180,E1 -8026.678,E2 -8026.678} C_VEL
LIN {X 0,Y 464.267,Z 137.237,A -85,B 0,C 180,E1 -8026.836,E2 -8026.836} C_VEL
LIN {X 0,Y 460.928,Z 118.099,A -85,B 0,C 180,E1 -8027.276,E2 -8027.276} C_VEL
LIN {X 0,Y 460.919,Z 116.74,A -85,B 0,C 180,E1 -8027.446,E2 -8027.446} C_VEL
LIN {X 0,Y 461.563,Z 103.506,A -85,B 0,C 180,E1 -8030.5,E2 -8030.5} C_VEL
LIN {X 0,Y 462.328,Z 86.993,A -85,B 0,C 180,E1 -8034.205,E2 -8034.205} C_VEL
LIN {X 0,Y 462.38,Z 82.736,A -85,B 0,C 180,E1 -8035.188,E2 -8035.188} C_VEL
LIN {X 0,Y 460.623,Z 72.656,A -85,B 0,C 180,E1 -8037.755,E2 -8037.755} C_VEL
LIN {X 0,Y 460.524,Z 72.622,A -85,B 0,C 180,E1 -8041.283,E2 -8041.283} C_VEL
LIN {X 0,Y 460.536,Z 72.614,A -85,B 0,C 180,E1 -8044.505,E2 -8044.505} C_VEL
LIN {X 0,Y 460.53,Z 72.623,A -85,B 0,C 180,E1 -8047.62,E2 -8047.62} C_VEL
LIN {X 0,Y 460.541,Z 72.604,A -85,B 0,C 180,E1 -8050.269,E2 -8050.269} C_VEL
LIN {X 0,Y 460.501,Z 72.626,A -85,B 0,C 180,E1 -8053.375,E2 -8053.375} C_VEL
LIN {X 0,Y 460.5,Z 72.62,A -85,B 0,C 180,E1 -8056.624,E2 -8056.624} C_VEL
LIN {X 0,Y 460.54,Z 72.611,A -85,B 0,C 180,E1 -8059.731,E2 -8059.731} C_VEL
LIN {X 0,Y 460.501,Z 72.62,A -85,B 0,C 180,E1 -8062.523,E2 -8062.523} C_VEL
LIN {X 0,Y 460.548,Z 72.606,A -85,B 0,C 180,E1 -8065.623,E2 -8065.623} C_VEL
LIN {X 0,Y 460.538,Z 72.618,A -85,B 0,C 180,E1 -8068.744,E2 -8068.744} C_VEL
LIN {X 0,Y 460.582,Z 72.603,A -85,B 0,C 180,E1 -8072.253,E2 -8072.253} C_VEL
LIN {X 0,Y 460.56,Z 72.609,A -85,B 0,C 180,E1 -8074.705,E2 -8074.705} C_VEL
LIN {X 0,Y 460.512,Z 72.617,A -85,B 0,C 180,E1 -8077.571,E2 -8077.571} C_VEL
LIN {X 0,Y 460.57,Z 72.603,A -85,B 0,C 180,E1 -8080.384,E2 -8080.384} C_VEL
LIN {X 0,Y 460.565,Z 72.607,A -85,B 0,C 180,E1 -8083.146,E2 -8083.146} C_VEL
LIN {X 0,Y 460.555,Z 72.613,A -85,B 0,C 180,E1 -8085.867,E2 -8085.867} C_VEL
LIN {X 0,Y 460.611,Z 72.598,A -85,B 0,C 180,E1 -8088.559,E2 -8088.559} C_VEL
LIN {X 0,Y 460.695,Z 72.589,A -85,B 0,C 180,E1 -8092.108,E2 -8092.108} C_VEL
LIN {X 0,Y 460.697,Z 72.596,A -85,B 0,C 180,E1 -8094.748,E2 -8094.748} C_VEL
LIN {X 0,Y 460.8,Z 72.58,A -85,B 0,C 180,E1 -8097.377,E2 -8097.377} C_VEL
LIN {X 0,Y 460.852,Z 72.563,A -85,B 0,C 180,E1 -8100,E2 -8100} C_VEL
LIN {X 0,Y 460.8,Z 72.579,A -85,B 0,C 180,E1 -8102.622,E2 -8102.622} C_VEL
LIN {X 0,Y 460.709,Z 72.594,A -85,B 0,C 180,E1 -8106.129,E2 -8106.129} C_VEL
LIN {X 0,Y 460.628,Z 72.592,A -85,B 0,C 180,E1 -8108.776,E2 -8108.776} C_VEL
LIN {X 0,Y 460.633,Z 72.6,A -85,B 0,C 180,E1 -8112.456,E2 -8112.456} C_VEL
LIN {X 0,Y 460.599,Z 72.606,A -85,B 0,C 180,E1 -8115.997,E2 -8115.997} C_VEL
LIN {X 0,Y 460.569,Z 72.601,A -85,B 0,C 180,E1 -8118.901,E2 -8118.901} C_VEL
LIN {X 0,Y 460.514,Z 72.622,A -85,B 0,C 180,E1 -8121.485,E2 -8121.485} C_VEL
LIN {X 0,Y 460.541,Z 72.614,A -85,B 0,C 180,E1 -8124.332,E2 -8124.332} C_VEL
LIN {X 0,Y 460.577,Z 72.603,A -85,B 0,C 180,E1 -8127.243,E2 -8127.243} C_VEL
LIN {X 0,Y 460.509,Z 72.618,A -85,B 0,C 180,E1 -8130.24,E2 -8130.24} C_VEL
LIN {X 0,Y 460.527,Z 72.611,A -85,B 0,C 180,E1 -8133.324,E2 -8133.324} C_VEL
LIN {X 0,Y 460.476,Z 72.624,A -85,B 0,C 180,E1 -8136.529,E2 -8136.529} C_VEL
LIN {X 0,Y 460.57,Z 72.608,A -85,B 0,C 180,E1 -8139.858,E2 -8139.858} C_VEL
LIN {X 0,Y 460.51,Z 72.622,A -85,B 0,C 180,E1 -8142.9,E2 -8142.9} C_VEL
LIN {X 0,Y 460.506,Z 72.615,A -85,B 0,C 180,E1 -8145.83,E2 -8145.83} C_VEL
LIN {X 0,Y 460.528,Z 72.605,A -85,B 0,C 180,E1 -8148.989,E2 -8148.989} C_VEL
LIN {X 0,Y 460.523,Z 72.617,A -85,B 0,C 180,E1 -8151.267,E2 -8151.267} C_VEL
LIN {X 0,Y 460.51,Z 72.606,A -85,B 0,C 180,E1 -8154.554,E2 -8154.554} C_VEL
LIN {X 0,Y 460.528,Z 72.618,A -85,B 0,C 180,E1 -8157.715,E2 -8157.715} C_VEL
LIN {X 0,Y 460.536,Z 72.607,A -85,B 0,C 180,E1 -8160.769,E2 -8160.769} C_VEL
LIN {X 0,Y 460.56,Z 72.619,A -85,B 0,C 180,E1 -8163.735,E2 -8163.735} C_VEL
LIN {X 0,Y 460.543,Z 72.617,A -85,B 0,C 180,E1 -8166.624,E2 -8166.624} C_VEL
LIN {X 0,Y 460.549,Z 72.62,A -85,B 0,C 180,E1 -8169.453,E2 -8169.453} C_VEL
LIN {X 0,Y 460.556,Z 72.616,A -85,B 0,C 180,E1 -8172.23,E2 -8172.23} C_VEL
LIN {X 0,Y 460.564,Z 72.617,A -85,B 0,C 180,E1 -8174.965,E2 -8174.965} C_VEL
LIN {X 0,Y 460.608,Z 72.61,A -85,B 0,C 180,E1 -8178.559,E2 -8178.559} C_VEL
LIN {X 0,Y 460.574,Z 72.615,A -85,B 0,C 180,E1 -8179.22,E2 -8179.22} C_VEL
LIN {X 0,Y 459.919,Z 72.701,A -85,B 0,C 180,E1 -8179.95,E2 -8179.95} C_VEL
LIN {X 0,Y 457.102,Z 73.054,A -85,B 0,C 180,E1 -8181.137,E2 -8181.137} C_VEL
LIN {X 0,Y 454.723,Z 73.348,A -85,B 0,C 180,E1 -8182.094,E2 -8182.094} C_VEL
LIN {X 0,Y 453.711,Z 73.471,A -85,B 0,C 180,E1 -8182.833,E2 -8182.833} C_VEL
LIN {X 0,Y 453.634,Z 73.479,A -85,B 0,C 180,E1 -8183.083,E2 -8183.083} C_VEL
LIN {X 0,Y 453.67,Z 73.476,A -85,B 0,C 180,E1 -8184.667,E2 -8184.667} C_VEL
LIN {X 0,Y 453.762,Z 73.465,A -85,B 0,C 180,E1 -8187.337,E2 -8187.337} C_VEL
LIN {X 0,Y 453.821,Z 73.456,A -85,B 0,C 180,E1 -8190,E2 -8190} C_VEL
LIN {X 0,Y 453.762,Z 73.465,A -85,B 0,C 180,E1 -8192.663,E2 -8192.663} C_VEL
LIN {X 0,Y 453.676,Z 73.475,A -85,B 0,C 180,E1 -8196.225,E2 -8196.225} C_VEL
LIN {X 0,Y 453.589,Z 73.487,A -85,B 0,C 180,E1 -8198.913,E2 -8198.913} C_VEL
LIN {X 0,Y 453.56,Z 73.491,A -85,B 0,C 180,E1 -8202.529,E2 -8202.529} C_VEL
LIN {X 0,Y 453.541,Z 73.493,A -85,B 0,C 180,E1 -8206.196,E2 -8206.196} C_VEL
LIN {X 0,Y 453.517,Z 73.493,A -85,B 0,C 180,E1 -8209.041,E2 -8209.041} C_VEL
LIN {X 0,Y 453.473,Z 73.5,A -85,B 0,C 180,E1 -8211.836,E2 -8211.836} C_VEL
LIN {X 0,Y 453.511,Z 73.494,A -85,B 0,C 180,E1 -8214.734,E2 -8214.734} C_VEL
LIN {X 0,Y 453.534,Z 73.489,A -85,B 0,C 180,E1 -8217.961,E2 -8217.961} C_VEL
LIN {X 0,Y 453.463,Z 73.499,A -85,B 0,C 180,E1 -8221.526,E2 -8221.526} C_VEL
LIN {X 0,Y 453.486,Z 73.474,A -85,B 0,C 180,E1 -8224.778,E2 -8224.778} C_VEL
LIN {X 0,Y 453.47,Z 73.497,A -85,B 0,C 180,E1 -8228.311,E2 -8228.311} C_VEL
LIN {X 0,Y 453.49,Z 73.482,A -85,B 0,C 180,E1 -8230.609,E2 -8230.609} C_VEL
LIN {X 0,Y 453.449,Z 73.48,A -85,B 0,C 180,E1 -8233.244,E2 -8233.244} C_VEL
LIN {X 0,Y 453.463,Z 73.501,A -85,B 0,C 180,E1 -8235.779,E2 -8235.779} C_VEL
LIN {X 0,Y 453.513,Z 73.488,A -85,B 0,C 180,E1 -8239.406,E2 -8239.406} C_VEL
LIN {X 0,Y 453.473,Z 73.496,A -85,B 0,C 180,E1 -8242.223,E2 -8242.223} C_VEL
LIN {X 0,Y 453.486,Z 73.489,A -85,B 0,C 180,E1 -8245.223,E2 -8245.223} C_VEL
LIN {X 0,Y 453.463,Z 73.497,A -85,B 0,C 180,E1 -8248.475,E2 -8248.475} C_VEL
LIN {X 0,Y 453.535,Z 73.478,A -85,B 0,C 180,E1 -8252.04,E2 -8252.04} C_VEL
LIN {X 0,Y 453.512,Z 73.492,A -85,B 0,C 180,E1 -8255.266,E2 -8255.266} C_VEL
LIN {X 0,Y 453.478,Z 73.497,A -85,B 0,C 180,E1 -8258.415,E2 -8258.415} C_VEL
LIN {X 0,Y 453.52,Z 73.478,A -85,B 0,C 180,E1 -8261.009,E2 -8261.009} C_VEL
LIN {X 0,Y 453.567,Z 73.481,A -85,B 0,C 180,E1 -8263.88,E2 -8263.88} C_VEL
LIN {X 0,Y 453.601,Z 73.475,A -85,B 0,C 180,E1 -8267.473,E2 -8267.473} C_VEL
LIN {X 0,Y 453.591,Z 73.469,A -85,B 0,C 180,E1 -8271.087,E2 -8271.087} C_VEL
LIN {X 0,Y 453.677,Z 73.469,A -85,B 0,C 180,E1 -8273.775,E2 -8273.775} C_VEL
LIN {X 0,Y 453.744,Z 73.457,A -85,B 0,C 180,E1 -8277.337,E2 -8277.337} C_VEL
LIN {X 0,Y 453.822,Z 73.438,A -85,B 0,C 180,E1 -8280,E2 -8280} C_VEL
LIN {X 0,Y 453.744,Z 73.459,A -85,B 0,C 180,E1 -8282.664,E2 -8282.664} C_VEL
LIN {X 0,Y 453.678,Z 73.469,A -85,B 0,C 180,E1 -8286.226,E2 -8286.226} C_VEL
LIN {X 0,Y 453.592,Z 73.467,A -85,B 0,C 180,E1 -8288.914,E2 -8288.914} C_VEL
LIN {X 0,Y 453.564,Z 73.48,A -85,B 0,C 180,E1 -8292.529,E2 -8292.529} C_VEL
LIN {X 0,Y 453.545,Z 73.481,A -85,B 0,C 180,E1 -8296.196,E2 -8296.196} C_VEL
LIN {X 0,Y 453.521,Z 73.475,A -85,B 0,C 180,E1 -8299.041,E2 -8299.041} C_VEL
LIN {X 0,Y 453.477,Z 73.495,A -85,B 0,C 180,E1 -8301.837,E2 -8301.837} C_VEL
LIN {X 0,Y 453.515,Z 73.49,A -85,B 0,C 180,E1 -8304.735,E2 -8304.735} C_VEL
LIN {X 0,Y 453.533,Z 73.48,A -85,B 0,C 180,E1 -8307.96,E2 -8307.96} C_VEL
LIN {X 0,Y 453.467,Z 73.496,A -85,B 0,C 180,E1 -8311.525,E2 -8311.525} C_VEL
LIN {X 0,Y 453.489,Z 73.487,A -85,B 0,C 180,E1 -8314.778,E2 -8314.778} C_VEL
LIN {X 0,Y 453.462,Z 73.499,A -85,B 0,C 180,E1 -8318.312,E2 -8318.312} C_VEL
LIN {X 0,Y 453.495,Z 73.49,A -85,B 0,C 180,E1 -8320.609,E2 -8320.609} C_VEL
LIN {X 0,Y 453.456,Z 73.498,A -85,B 0,C 180,E1 -8323.244,E2 -8323.244} C_VEL
LIN {X 0,Y 453.465,Z 73.495,A -85,B 0,C 180,E1 -8325.779,E2 -8325.779} C_VEL
LIN {X 0,Y 453.481,Z 73.495,A -85,B 0,C 180,E1 -8328.21,E2 -8328.21} C_VEL
LIN {X 0,Y 453.493,Z 73.488,A -85,B 0,C 180,E1 -8330.794,E2 -8330.794} C_VEL
LIN {X 0,Y 453.459,Z 73.497,A -85,B 0,C 180,E1 -8333.918,E2 -8333.918} C_VEL
LIN {X 0,Y 453.485,Z 73.494,A -85,B 0,C 180,E1 -8337.152,E2 -8337.152} C_VEL
LIN {X 0,Y 453.477,Z 73.495,A -85,B 0,C 180,E1 -8340.269,E2 -8340.269} C_VEL
LIN {X 0,Y 453.594,Z 73.652,A -85,B 0,C 180,E1 -8342.08,E2 -8342.08} C_VEL
LIN {X 0,Y 455.387,Z 83.633,A -85,B 0,C 180,E1 -8344.642,E2 -8344.642} C_VEL
LIN {X 0,Y 455.286,Z 89.098,A -85,B 0,C 180,E1 -8345.962,E2 -8345.962} C_VEL
LIN {X 0,Y 454.506,Z 105.197,A -85,B 0,C 180,E1 -8349.64,E2 -8349.64} C_VEL
LIN {X 0,Y 453.911,Z 117.251,A -85,B 0,C 180,E1 -8352.397,E2 -8352.397} C_VEL
LIN {X 0,Y 454.415,Z 120.542,A -85,B 0,C 180,E1 -8352.521,E2 -8352.521} C_VEL
LIN {X 0,Y 457.569,Z 139.025,A -85,B 0,C 180,E1 -8352.941,E2 -8352.941} C_VEL
LIN {X 0,Y 456.868,Z 222.143,A -85,B 0,C 180,E1 -8354.269,E2 -8354.269} C_VEL
LIN {X 0,Y 456.618,Z 232.04,A -85,B 0,C 180,E1 -8354.517,E2 -8354.517} C_VEL
LIN {X 0,Y 456.282,Z 242.017,A -85,B 0,C 180,E1 -8354.878,E2 -8354.878} C_VEL
LIN {X 0,Y 455.854,Z 252.381,A -85,B 0,C 180,E1 -8355.377,E2 -8355.377} C_VEL
LIN {X 0,Y 455.414,Z 261.517,A -85,B 0,C 180,E1 -8355.933,E2 -8355.933} C_VEL
LIN {X 0,Y 454.924,Z 270.514,A -85,B 0,C 180,E1 -8356.601,E2 -8356.601} C_VEL
LIN {X 0,Y 454.492,Z 278.99,A -85,B 0,C 180,E1 -8357.358,E2 -8357.358} C_VEL
LIN {X 0,Y 454.108,Z 286.642,A -85,B 0,C 180,E1 -8358.167,E2 -8358.167} C_VEL
LIN {X 0,Y 453.686,Z 293.862,A -85,B 0,C 180,E1 -8359.061,E2 -8359.061} C_VEL
LIN {X 0,Y 453.363,Z 300.065,A -85,B 0,C 180,E1 -8359.956,E2 -8359.956} C_VEL
LIN {X 0,Y 453.037,Z 306.602,A -85,B 0,C 180,E1 -8361.076,E2 -8361.076} C_VEL
LIN {X 0,Y 452.846,Z 311.103,A -85,B 0,C 180,E1 -8361.971,E2 -8361.971} C_VEL
LIN {X 0,Y 452.644,Z 316.749,A -85,B 0,C 180,E1 -8363.358,E2 -8363.358} C_VEL
LIN {X 0,Y 452.559,Z 320.916,A -85,B 0,C 180,E1 -8364.654,E2 -8364.654} C_VEL
LIN {X 0,Y 452.486,Z 323.28,A -85,B 0,C 180,E1 -8365.546,E2 -8365.546} C_VEL
LIN {X 0,Y 452.48,Z 325.077,A -85,B 0,C 180,E1 -8366.438,E2 -8366.438} C_VEL
LIN {X 0,Y 452.437,Z 327.517,A -85,B 0,C 180,E1 -8368.22,E2 -8368.22} C_VEL
LIN {X 0,Y 452.431,Z 328.105,A -85,B 0,C 180,E1 -8369.11,E2 -8369.11} C_VEL
LIN {X 0,Y 452.431,Z 328.105,A -85,B 0,C 180,E1 -8370.89,E2 -8370.89} C_VEL
LIN {X 0,Y 452.437,Z 327.517,A -85,B 0,C 180,E1 -8371.78,E2 -8371.78} C_VEL
LIN {X 0,Y 452.48,Z 325.077,A -85,B 0,C 180,E1 -8373.562,E2 -8373.562} C_VEL
LIN {X 0,Y 452.544,Z 322.132,A -85,B 0,C 180,E1 -8374.9,E2 -8374.9} C_VEL
LIN {X 0,Y 452.585,Z 318.146,A -85,B 0,C 180,E1 -8376.24,E2 -8376.24} C_VEL
LIN {X 0,Y 452.738,Z 313.018,A -85,B 0,C 180,E1 -8377.582,E2 -8377.582} C_VEL
LIN {X 0,Y 453.002,Z 307.758,A -85,B 0,C 180,E1 -8378.7,E2 -8378.7} C_VEL
LIN {X 0,Y 453.292,Z 301.441,A -85,B 0,C 180,E1 -8379.82,E2 -8379.82} C_VEL
LIN {X 0,Y 453.582,Z 295.489,A -85,B 0,C 180,E1 -8380.715,E2 -8380.715} C_VEL
LIN {X 0,Y 453.989,Z 288.561,A -85,B 0,C 180,E1 -8381.61,E2 -8381.61} C_VEL
LIN {X 0,Y 454.434,Z 280.38,A -85,B 0,C 180,E1 -8382.504,E2 -8382.504} C_VEL
LIN {X 0,Y 454.865,Z 272.378,A -85,B 0,C 180,E1 -8383.244,E2 -8383.244} C_VEL
LIN {X 0,Y 455.318,Z 263.148,A -85,B 0,C 180,E1 -8383.956,E2 -8383.956} C_VEL
LIN {X 0,Y 455.793,Z 253.388,A -85,B 0,C 180,E1 -8384.568,E2 -8384.568} C_VEL
LIN {X 0,Y 456.189,Z 244.593,A -85,B 0,C 180,E1 -8385.011,E2 -8385.011} C_VEL
LIN {X 0,Y 456.57,Z 234.664,A -85,B 0,C 180,E1 -8385.398,E2 -8385.398} C_VEL
LIN {X 0,Y 456.862,Z 224.808,A -85,B 0,C 180,E1 -8385.674,E2 -8385.674} C_VEL
LIN {X 0,Y 457.142,Z 200.774,A -85,B 0,C 180,E1 -8386.084,E2 -8386.084} C_VEL
LIN {X 0,Y 457.469,Z 138.162,A -85,B 0,C 180,E1 -8387.076,E2 -8387.076} C_VEL
LIN {X 0,Y 453.966,Z 117.713,A -85,B 0,C 180,E1 -8387.558,E2 -8387.558} C_VEL
LIN {X 0,Y 453.928,Z 116.69,A -85,B 0,C 180,E1 -8387.692,E2 -8387.692} C_VEL
LIN {X 0,Y 454.608,Z 103.345,A -85,B 0,C 180,E1 -8390.828,E2 -8390.828} C_VEL
LIN {X 0,Y 455.313,Z 89.283,A -85,B 0,C 180,E1 -8394.041,E2 -8394.041} C_VEL
LIN {X 0,Y 455.371,Z 83.633,A -85,B 0,C 180,E1 -8395.358,E2 -8395.358} C_VEL
LIN {X 0,Y 453.574,Z 73.557,A -85,B 0,C 180,E1 -8397.969,E2 -8397.969} C_VEL
LIN {X 0,Y 453.468,Z 73.498,A -85,B 0,C 180,E1 -8401.525,E2 -8401.525} C_VEL
LIN {X 0,Y 453.491,Z 73.491,A -85,B 0,C 180,E1 -8404.777,E2 -8404.777} C_VEL
LIN {X 0,Y 453.473,Z 73.494,A -85,B 0,C 180,E1 -8408.311,E2 -8408.311} C_VEL
LIN {X 0,Y 453.496,Z 73.481,A -85,B 0,C 180,E1 -8410.609,E2 -8410.609} C_VEL
LIN {X 0,Y 453.457,Z 73.502,A -85,B 0,C 180,E1 -8413.244,E2 -8413.244} C_VEL
LIN {X 0,Y 453.465,Z 73.499,A -85,B 0,C 180,E1 -8415.778,E2 -8415.778} C_VEL
LIN {X 0,Y 453.48,Z 73.494,A -85,B 0,C 180,E1 -8418.209,E2 -8418.209} C_VEL
LIN {X 0,Y 453.489,Z 73.49,A -85,B 0,C 180,E1 -8420.794,E2 -8420.794} C_VEL
LIN {X 0,Y 453.456,Z 73.495,A -85,B 0,C 180,E1 -8423.917,E2 -8423.917} C_VEL
LIN {X 0,Y 453.484,Z 73.494,A -85,B 0,C 180,E1 -8427.151,E2 -8427.151} C_VEL
LIN {X 0,Y 453.476,Z 73.495,A -85,B 0,C 180,E1 -8430.268,E2 -8430.268} C_VEL
LIN {X 0,Y 453.507,Z 73.483,A -85,B 0,C 180,E1 -8433.294,E2 -8433.294} C_VEL
LIN {X 0,Y 453.505,Z 73.491,A -85,B 0,C 180,E1 -8436.238,E2 -8436.238} C_VEL
LIN {X 0,Y 453.483,Z 73.488,A -85,B 0,C 180,E1 -8439.117,E2 -8439.117} C_VEL
LIN {X 0,Y 453.511,Z 73.475,A -85,B 0,C 180,E1 -8441.944,E2 -8441.944} C_VEL
LIN {X 0,Y 453.54,Z 73.489,A -85,B 0,C 180,E1 -8444.726,E2 -8444.726} C_VEL
LIN {X 0,Y 453.56,Z 73.478,A -85,B 0,C 180,E1 -8448.379,E2 -8448.379} C_VEL
LIN {X 0,Y 453.652,Z 73.464,A -85,B 0,C 180,E1 -8451.985,E2 -8451.985} C_VEL
